C03629=1083.943,283.313,-84.249,175.955,24.447,154.018
C03630=1083.938,283.065,-84.220,175.952,24.443,154.018
C03631=1083.932,282.817,-84.190,175.949,24.440,154.017
C03632=1083.926,282.569,-84.160,175.947,24.436,154.017
C03633=1083.920,282.321,-84.131,175.944,24.433,154.016
C03634=1083.915,282.073,-84.101,175.941,24.429,154.016
C03635=1083.910,281.824,-84.072,175.938,24.426,154.015
C03636=1083.903,281.576,-84.043,175.936,24.423,154.015
C03637=1083.898,281.328,-84.013,175.933,24.419,154.015
C03638=1083.892,281.079,-83.984,175.930,24.415,154.014
C03639=1083.886,280.831,-83.954,175.927,24.412,154.014
C03640=1083.881,280.584,-83.925,175.925,24.409,154.013
C03641=1083.875,280.335,-83.896,175.922,24.405,154.013
C03642=1083.870,280.087,-83.867,175.919,24.402,154.013
C03643=1083.863,279.839,-83.837,175.916,24.398,154.012
C03644=1083.858,279.590,-83.808,175.913,24.395,154.012
C03645=1083.852,279.342,-83.778,175.910,24.391,154.011
C03646=1083.846,279.094,-83.749,175.907,24.388,154.011
C03647=1083.841,278.846,-83.720,175.904,24.384,154.011
C03648=1083.835,278.598,-83.691,175.902,24.381,154.010
C03649=1083.829,278.350,-83.661,175.899,24.378,154.010
C03650=1083.823,278.101,-83.632,175.896,24.374,154.009
C03651=1083.818,277.853,-83.603,175.893,24.370,154.009
C03652=1083.812,277.606,-83.574,175.891,24.367,154.009
C03653=1083.807,277.356,-83.545,175.888,24.364,154.008
C03654=1083.800,277.108,-83.516,175.885,24.360,154.008
C03655=1083.791,276.725,-83.471,175.881,24.355,154.007
C03656=1083.783,276.341,-83.426,175.877,24.350,154.007
C03657=1083.773,275.957,-83.380,175.872,24.345,154.006
C03658=1083.765,275.574,-83.336,175.868,24.339,154.005
C03659=1083.760,275.325,-83.307,175.865,24.336,154.005
C03660=1083.753,275.077,-83.278,175.863,24.333,154.005
C03661=1083.748,274.829,-83.249,175.860,24.329,154.004
C03662=1083.743,274.581,-83.221,175.857,24.325,154.004
C03663=1083.736,274.333,-83.192,175.854,24.322,154.003
C03664=1083.731,274.084,-83.162,175.852,24.319,154.003
C03665=1083.726,273.836,-83.134,175.849,24.315,154.003
C03666=1083.719,273.588,-83.105,175.846,24.312,154.002
C03667=1083.714,273.339,-83.075,175.843,24.309,154.002
C03668=1083.708,273.091,-83.047,175.840,24.305,154.001
C03669=1083.702,272.843,-83.018,175.837,24.302,154.001
C03670=1083.697,272.594,-82.989,175.835,24.299,154.001
C03671=1083.691,272.346,-82.960,175.832,24.295,154.000
C03672=1083.685,272.099,-82.932,175.829,24.291,154.000
C03673=1083.679,271.850,-82.903,175.826,24.288,153.999
C03674=1083.674,271.601,-82.874,175.824,24.285,153.999
C03675=1083.668,271.353,-82.846,175.821,24.282,153.999
C03676=1083.662,271.105,-82.817,175.818,24.278,153.998
C03677=1083.656,270.857,-82.788,175.816,24.275,153.998
C03678=1083.651,270.609,-82.760,175.813,24.271,153.998
C03679=1083.645,270.360,-82.731,175.810,24.268,153.997
C03680=1083.639,270.111,-82.702,175.808,24.265,153.997
C03681=1083.634,269.864,-82.674,175.804,24.262,153.996
C03682=1083.628,269.615,-82.645,175.801,24.258,153.996
C03683=1083.621,269.367,-82.616,175.799,24.255,153.996
C03684=1083.617,269.119,-82.588,175.796,24.251,153.995
C03685=1083.611,268.870,-82.560,175.793,24.248,153.995
C03686=1083.605,268.622,-82.531,175.791,24.245,153.995
C03687=1083.599,268.374,-82.503,175.788,24.241,153.994
C03688=1083.593,268.125,-82.474,175.785,24.238,153.994
C03689=1083.588,267.878,-82.446,175.782,24.234,153.993
C03690=1083.582,267.629,-82.417,175.780,24.231,153.993
C03691=1083.576,267.381,-82.389,175.777,24.228,153.993
C03692=1083.570,267.132,-82.361,175.774,24.224,153.992
C03693=1083.564,266.884,-82.332,175.772,24.221,153.992
C03694=1083.559,266.636,-82.304,175.769,24.218,153.991
C03695=1083.553,266.387,-82.276,175.766,24.215,153.991
C03696=1083.548,266.139,-82.248,175.763,24.211,153.991
C03697=1083.542,265.891,-82.218,175.760,24.208,153.990
C03698=1083.537,265.642,-82.190,175.758,24.205,153.990
C03699=1083.531,265.394,-82.162,175.755,24.201,153.990
C03700=1083.525,265.146,-82.134,175.752,24.198,153.989
C03701=1083.520,264.897,-82.105,175.750,24.195,153.989
C03702=1083.514,264.649,-82.077,175.747,24.191,153.988
C03703=1083.508,264.400,-82.049,175.744,24.188,153.988
C03704=1083.503,264.153,-82.020,175.742,24.184,153.988
C03705=1083.497,263.904,-81.992,175.739,24.181,153.987
C03706=1083.490,263.656,-81.964,175.736,24.178,153.987
C03707=1083.482,263.274,-81.921,175.732,24.173,153.987
C03708=1083.473,262.894,-81.878,175.728,24.168,153.986
C03709=1083.464,262.513,-81.836,175.724,24.164,153.985
C03710=1083.455,262.133,-81.793,175.719,24.158,153.985
C03711=1083.449,261.884,-81.764,175.716,24.155,153.984
C03712=1083.444,261.636,-81.736,175.714,24.152,153.984
C03713=1083.437,261.387,-81.709,175.711,24.148,153.984
C03714=1083.431,261.139,-81.681,175.709,24.146,153.983
C03715=1083.426,260.890,-81.652,175.706,24.142,153.983
C03716=1083.419,260.643,-81.625,175.703,24.138,153.983
C03717=1083.414,260.393,-81.597,175.701,24.136,153.982
C03718=1083.408,260.145,-81.570,175.698,24.132,153.982
C03719=1083.403,259.897,-81.541,175.695,24.129,153.982
C03720=1083.396,259.649,-81.514,175.692,24.126,153.981
C03721=1083.391,259.400,-81.486,175.689,24.122,153.981
C03722=1083.385,259.152,-81.458,175.687,24.120,153.981
C03723=1083.379,258.903,-81.431,175.684,24.116,153.980
C03724=1083.373,258.655,-81.403,175.681,24.112,153.980
C03725=1083.368,258.407,-81.375,175.679,24.110,153.980
C03726=1083.362,258.158,-81.346,175.676,24.106,153.979
C03727=1083.356,257.910,-81.319,175.674,24.103,153.979
C03728=1083.350,257.661,-81.291,175.671,24.100,153.978
C03729=1083.345,257.413,-81.263,175.668,24.096,153.978
C03730=1083.339,257.165,-81.236,175.666,24.093,153.978
C03731=1083.333,256.916,-81.208,175.663,24.090,153.977
C03732=1083.328,256.668,-81.180,175.660,24.087,153.977
C03733=1083.321,256.419,-81.153,175.657,24.083,153.977
C03734=1083.316,256.171,-81.125,175.654,24.080,153.976
C03735=1083.310,255.923,-81.098,175.652,24.077,153.976
C03736=1083.304,255.674,-81.070,175.649,24.074,153.976
C03737=1083.299,255.426,-81.043,175.647,24.071,153.975
C03738=1083.293,255.178,-81.015,175.644,24.067,153.975
C03739=1083.288,254.928,-80.988,175.641,24.064,153.975
C03740=1083.282,254.680,-80.960,175.639,24.061,153.974
C03741=1083.276,254.433,-80.932,175.636,24.057,153.974
C03742=1083.270,254.183,-80.905,175.634,24.055,153.973
C03743=1083.264,253.936,-80.877,175.631,24.051,153.973
C03744=1083.259,253.687,-80.850,175.628,24.048,153.973
C03745=1083.253,253.438,-80.822,175.625,24.045,153.972
C03746=1083.248,253.190,-80.795,175.622,24.041,153.972
C03747=1083.242,252.942,-80.767,175.620,24.038,153.972
C03748=1083.237,252.693,-80.740,175.617,24.035,153.971
C03749=1083.231,252.445,-80.712,175.615,24.032,153.971
C03750=1083.226,252.196,-80.685,175.612,24.028,153.971
C03751=1083.220,251.948,-80.658,175.610,24.025,153.970
C03752=1083.214,251.699,-80.630,175.607,24.022,153.970
C03753=1083.208,251.450,-80.603,175.604,24.018,153.969
C03754=1083.203,251.202,-80.575,175.602,24.015,153.969
C03755=1083.197,250.954,-80.549,175.599,24.012,153.969
C03756=1083.192,250.705,-80.521,175.597,24.009,153.968
C03757=1083.186,250.458,-80.494,175.594,24.005,153.968
C03758=1083.180,250.208,-80.466,175.591,24.002,153.968
C03759=1083.172,249.825,-80.424,175.587,23.997,153.967
C03760=1083.163,249.441,-80.383,175.583,23.992,153.966
C03761=1083.155,249.058,-80.341,175.579,23.987,153.966
C03762=1083.146,248.674,-80.299,175.575,23.982,153.965
C03763=1083.140,248.426,-80.272,175.572,23.978,153.965
C03764=1083.135,248.177,-80.245,175.570,23.975,153.965
C03765=1083.129,247.929,-80.217,175.567,23.972,153.964
C03766=1083.123,247.680,-80.190,175.565,23.969,153.964
C03767=1083.118,247.432,-80.163,175.562,23.965,153.964
C03768=1083.113,247.183,-80.136,175.560,23.963,153.963
C03769=1083.107,246.935,-80.109,175.557,23.959,153.963
C03770=1083.101,246.686,-80.082,175.555,23.956,153.962
C03771=1083.096,246.438,-80.054,175.551,23.953,153.962
C03772=1083.089,246.189,-80.027,175.549,23.949,153.962
C03773=1083.084,245.941,-80.001,175.546,23.946,153.961
C03774=1083.079,245.692,-79.974,175.543,23.943,153.961
C03775=1083.073,245.444,-79.947,175.541,23.939,153.961
C03776=1083.067,245.195,-79.920,175.538,23.936,153.960
C03777=1083.062,244.947,-79.893,175.536,23.933,153.960
C03778=1083.056,244.698,-79.866,175.533,23.930,153.960
C03779=1083.050,244.450,-79.840,175.531,23.927,153.959
C03780=1083.045,244.202,-79.813,175.528,23.923,153.959
C03781=1083.039,243.952,-79.785,175.526,23.921,153.959
C03782=1083.033,243.704,-79.759,175.523,23.917,153.958
C03783=1083.028,243.455,-79.732,175.521,23.914,153.958
C03784=1083.022,243.207,-79.706,175.517,23.911,153.958
C03785=1083.017,242.958,-79.678,175.515,23.907,153.957
C03786=1083.011,242.710,-79.652,175.512,23.904,153.957
C03787=1083.005,242.462,-79.625,175.510,23.901,153.956
C03788=1082.999,242.213,-79.598,175.507,23.897,153.956
C03789=1082.994,241.965,-79.572,175.505,23.895,153.956
C03790=1082.988,241.716,-79.546,175.502,23.891,153.955
C03791=1082.982,241.468,-79.519,175.500,23.888,153.955
C03792=1082.976,241.219,-79.492,175.497,23.885,153.955
C03793=1082.970,240.970,-79.465,175.495,23.882,153.954
C03794=1082.964,240.722,-79.439,175.492,23.878,153.954
C03795=1082.959,240.473,-79.412,175.489,23.876,153.954
C03796=1082.954,240.224,-79.386,175.486,23.872,153.953
C03797=1082.948,239.976,-79.359,175.484,23.869,153.953
C03798=1082.942,239.728,-79.332,175.481,23.866,153.953
C03799=1082.937,239.479,-79.306,175.479,23.863,153.952
C03800=1082.931,239.230,-79.280,175.476,23.859,153.952
C03801=1082.925,238.982,-79.253,175.474,23.857,153.952
C03802=1082.920,238.733,-79.226,175.471,23.853,153.951
C03803=1082.914,238.485,-79.200,175.469,23.850,153.951
C03804=1082.908,238.236,-79.174,175.467,23.847,153.951
C03805=1082.903,237.988,-79.147,175.464,23.844,153.950
C03806=1082.897,237.739,-79.121,175.461,23.841,153.950
C03807=1082.891,237.490,-79.095,175.459,23.837,153.950
C03808=1082.886,237.242,-79.068,175.456,23.835,153.949
C03809=1082.880,236.993,-79.042,175.453,23.831,153.949
C03810=1082.874,236.745,-79.015,175.451,23.828,153.949
C03811=1082.866,236.354,-78.975,175.447,23.823,153.948
C03812=1082.856,235.964,-78.933,175.443,23.818,153.947
C03813=1082.847,235.574,-78.892,175.439,23.813,153.947
C03814=1082.839,235.183,-78.851,175.435,23.808,153.946
C03815=1082.832,234.935,-78.825,175.433,23.805,153.946
C03816=1082.827,234.686,-78.799,175.430,23.801,153.946
C03817=1082.821,234.438,-78.772,175.428,23.799,153.945
C03818=1082.816,234.189,-78.746,175.425,23.795,153.945
C03819=1082.810,233.940,-78.719,175.423,23.792,153.945
C03820=1082.805,233.692,-78.693,175.419,23.789,153.944
C03821=1082.799,233.443,-78.667,175.417,23.786,153.944
C03822=1082.794,233.195,-78.641,175.414,23.782,153.944
C03823=1082.788,232.946,-78.616,175.412,23.779,153.943
C03824=1082.782,232.698,-78.589,175.410,23.776,153.943
C03825=1082.776,232.449,-78.563,175.407,23.773,153.943
C03826=1082.771,232.201,-78.537,175.405,23.770,153.942
C03827=1082.765,231.952,-78.511,175.402,23.766,153.942
C03828=1082.759,231.703,-78.485,175.400,23.764,153.942
C03829=1082.753,231.454,-78.459,175.397,23.760,153.941
C03830=1082.748,231.206,-78.433,175.395,23.757,153.941
C03831=1082.743,230.957,-78.407,175.392,23.754,153.941
C03832=1082.737,230.708,-78.381,175.390,23.751,153.940
C03833=1082.731,230.460,-78.355,175.387,23.748,153.940
C03834=1082.725,230.211,-78.329,175.384,23.744,153.940
C03835=1082.720,229.962,-78.303,175.382,23.741,153.939
C03836=1082.714,229.715,-78.278,175.379,23.738,153.939
C03837=1082.709,229.466,-78.252,175.377,23.735,153.939
C03838=1082.703,229.217,-78.226,175.375,23.732,153.938
C03839=1082.697,228.968,-78.200,175.372,23.729,153.938
C03840=1082.691,228.719,-78.175,175.370,23.726,153.937
C03841=1082.685,228.471,-78.148,175.367,23.722,153.937
C03842=1082.679,228.222,-78.123,175.365,23.719,153.937
C03843=1082.675,227.974,-78.097,175.362,23.716,153.937
C03844=1082.668,227.725,-78.072,175.359,23.713,153.936
C03845=1082.663,227.476,-78.046,175.357,23.710,153.936
C03846=1082.657,227.228,-78.020,175.354,23.707,153.936
C03847=1082.651,226.979,-77.994,175.352,23.704,153.935
C03848=1082.646,226.731,-77.969,175.350,23.701,153.935
C03849=1082.640,226.482,-77.943,175.347,23.697,153.935
C03850=1082.634,226.233,-77.917,175.345,23.694,153.934
C03851=1082.628,225.985,-77.892,175.342,23.691,153.934
C03852=1082.623,225.736,-77.866,175.340,23.688,153.933
C03853=1082.617,225.488,-77.841,175.338,23.685,153.933
C03854=1082.612,225.239,-77.815,175.335,23.681,153.933
C03855=1082.605,224.990,-77.789,175.332,23.679,153.932
C03856=1082.601,224.742,-77.764,175.329,23.675,153.932
C03857=1082.594,224.493,-77.738,175.327,23.672,153.932
C03858=1082.589,224.244,-77.713,175.325,23.669,153.931
C03859=1082.583,223.996,-77.688,175.322,23.666,153.931
C03860=1082.578,223.747,-77.662,175.320,23.663,153.931
C03861=1082.572,223.499,-77.636,175.318,23.660,153.930
C03862=1082.566,223.249,-77.611,175.315,23.656,153.930
C03863=1082.557,222.851,-77.570,175.311,23.651,153.929
C03864=1082.549,222.452,-77.529,175.307,23.646,153.929
C03865=1082.540,222.053,-77.489,175.303,23.641,153.928
C03866=1082.530,221.654,-77.448,175.300,23.636,153.928
C03867=1082.525,221.406,-77.423,175.297,23.633,153.928
C03868=1082.519,221.157,-77.397,175.294,23.630,153.927
C03869=1082.513,220.907,-77.372,175.292,23.627,153.927
C03870=1082.508,220.660,-77.347,175.289,23.624,153.927
C03871=1082.501,220.411,-77.322,175.287,23.621,153.926
C03872=1082.496,220.162,-77.296,175.284,23.618,153.926
C03873=1082.491,219.913,-77.272,175.282,23.614,153.926
C03874=1082.484,219.665,-77.246,175.280,23.612,153.925
C03875=1082.479,219.416,-77.221,175.277,23.608,153.925
C03876=1082.473,219.168,-77.196,175.275,23.605,153.925
C03877=1082.468,218.918,-77.171,175.273,23.602,153.924
C03878=1082.461,218.670,-77.146,175.270,23.599,153.924
C03879=1082.456,218.421,-77.120,175.268,23.596,153.924
C03880=1082.451,218.172,-77.095,175.265,23.593,153.923
C03881=1082.445,217.924,-77.070,175.263,23.589,153.923
C03882=1082.439,217.676,-77.045,175.260,23.586,153.923
C03883=1082.434,217.426,-77.020,175.258,23.583,153.922
C03884=1082.428,217.178,-76.995,175.255,23.580,153.922
C03885=1082.422,216.929,-76.970,175.253,23.577,153.921
C03886=1082.416,216.681,-76.945,175.251,23.574,153.921
C03887=1082.411,216.432,-76.919,175.248,23.570,153.921
C03888=1082.406,216.183,-76.895,175.246,23.568,153.921
C03889=1082.399,215.934,-76.870,175.244,23.564,153.920
C03890=1082.394,215.685,-76.845,175.241,23.561,153.920
C03891=1082.388,215.437,-76.820,175.239,23.558,153.919
C03892=1082.383,215.188,-76.795,175.236,23.555,153.919
C03893=1082.377,214.940,-76.770,175.234,23.552,153.919
C03894=1082.371,214.690,-76.745,175.231,23.549,153.919
C03895=1082.366,214.442,-76.720,175.229,23.546,153.918
C03896=1082.360,214.193,-76.696,175.226,23.542,153.918
C03897=1082.355,213.945,-76.670,175.224,23.539,153.917
C03898=1082.349,213.696,-76.646,175.222,23.536,153.917
C03899=1082.343,213.448,-76.621,175.219,23.533,153.917
C03900=1082.338,213.198,-76.596,175.217,23.530,153.916
C03901=1082.332,212.950,-76.572,175.215,23.527,153.916
C03902=1082.326,212.701,-76.546,175.212,23.523,153.916
C03903=1082.321,212.452,-76.522,175.210,23.520,153.915
C03904=1082.315,212.204,-76.497,175.208,23.517,153.915
C03905=1082.309,211.955,-76.473,175.205,23.514,153.915
C03906=1082.303,211.706,-76.448,175.203,23.511,153.914
C03907=1082.298,211.458,-76.423,175.200,23.508,153.914
C03908=1082.293,211.208,-76.398,175.198,23.505,153.914
C03909=1082.287,210.960,-76.373,175.195,23.502,153.913
C03910=1082.282,210.711,-76.349,175.193,23.498,153.913
C03911=1082.276,210.462,-76.324,175.191,23.496,153.913
C03912=1082.270,210.214,-76.300,175.188,23.492,153.912
C03913=1082.264,209.965,-76.276,175.186,23.489,153.912
C03914=1082.258,209.717,-76.251,175.184,23.486,153.912
C03915=1082.250,209.321,-76.212,175.180,23.481,153.911
C03916=1082.241,208.926,-76.173,175.176,23.476,153.911
C03917=1082.232,208.532,-76.134,175.172,23.471,153.910
C03918=1082.222,208.137,-76.095,175.169,23.466,153.910
C03919=1082.199,207.105,-75.995,175.076,23.417,153.912
C03920=1082.193,206.857,-75.972,175.073,23.415,153.912
C03921=1082.188,206.608,-75.947,175.071,23.413,153.912
C03922=1082.182,206.358,-75.923,175.068,23.411,153.911
C03923=1082.176,206.110,-75.900,175.065,23.408,153.911
C03924=1082.171,205.861,-75.875,175.063,23.406,153.911
C03925=1082.166,205.612,-75.852,175.060,23.404,153.911
C03926=1082.160,205.364,-75.828,175.058,23.402,153.911
C03927=1082.155,205.115,-75.804,175.056,23.399,153.911
C03928=1082.149,204.866,-75.779,175.053,23.397,153.911
C03929=1082.143,204.617,-75.756,175.051,23.395,153.911
C03930=1082.138,204.369,-75.732,175.048,23.393,153.910
C03931=1082.132,204.120,-75.708,175.046,23.391,153.910
C03932=1082.127,203.871,-75.685,175.044,23.389,153.910
C03933=1082.121,203.623,-75.661,175.040,23.386,153.910
C03934=1082.116,203.373,-75.637,175.038,23.384,153.910
C03935=1082.110,203.124,-75.613,175.036,23.382,153.910
C03936=1082.104,202.876,-75.589,175.033,23.380,153.910
C03937=1082.099,202.627,-75.566,175.031,23.378,153.910
C03938=1082.093,202.378,-75.542,175.028,23.375,153.910
C03939=1082.088,202.129,-75.519,175.026,23.373,153.909
C03940=1082.082,201.880,-75.494,175.024,23.371,153.909
C03941=1082.076,201.631,-75.471,175.021,23.369,153.909
C03942=1082.070,201.383,-75.447,175.019,23.367,153.909
C03943=1082.065,201.134,-75.424,175.016,23.365,153.909
C03944=1082.059,200.885,-75.400,175.014,23.363,153.909
C03945=1082.054,200.636,-75.377,175.012,23.361,153.909
C03946=1082.048,200.388,-75.353,175.009,23.358,153.909
C03947=1082.042,200.138,-75.330,175.006,23.356,153.909
C03948=1082.036,199.890,-75.306,175.003,23.354,153.909
C03949=1082.031,199.641,-75.283,175.001,23.352,153.908
C03950=1082.025,199.393,-75.259,174.999,23.350,153.908
C03951=1082.020,199.143,-75.235,174.996,23.348,153.908
C03952=1082.014,198.894,-75.212,174.994,23.346,153.908
C03953=1082.008,198.646,-75.189,174.992,23.343,153.908
C03954=1082.003,198.397,-75.165,174.989,23.342,153.908
C03955=1081.996,198.148,-75.141,174.987,23.339,153.908
C03956=1081.990,197.899,-75.118,174.984,23.337,153.908
C03957=1081.985,197.650,-75.095,174.982,23.335,153.908
C03958=1081.979,197.402,-75.071,174.979,23.333,153.907
C03959=1081.974,197.153,-75.048,174.977,23.331,153.907
C03960=1081.969,196.904,-75.025,174.975,23.329,153.907
C03961=1081.963,196.655,-75.001,174.972,23.327,153.907
C03962=1081.957,196.406,-74.978,174.970,23.325,153.907
C03963=1081.952,196.157,-74.954,174.967,23.322,153.907
C03964=1081.946,195.909,-74.931,174.965,23.320,153.907
C03965=1081.940,195.660,-74.908,174.963,23.319,153.907
C03966=1081.935,195.411,-74.884,174.960,23.316,153.907
C03967=1081.929,195.162,-74.861,174.958,23.314,153.906
C03968=1081.923,194.914,-74.838,174.956,23.312,153.906
C03969=1081.918,194.665,-74.815,174.953,23.310,153.906
C03970=1081.913,194.415,-74.791,174.951,23.308,153.906
C03971=1081.907,194.167,-74.768,174.948,23.306,153.906
C03972=1081.901,193.918,-74.745,174.946,23.303,153.906
C03973=1081.896,193.669,-74.721,174.944,23.301,153.906
C03974=1081.890,193.420,-74.698,174.941,23.299,153.906
C03975=1081.884,193.171,-74.675,174.939,23.297,153.906
C03976=1081.879,192.922,-74.652,174.936,23.295,153.905
C03977=1081.874,192.673,-74.629,174.934,23.293,153.905
C03978=1081.868,192.424,-74.606,174.932,23.291,153.905
C03979=1081.862,192.175,-74.583,174.929,23.289,153.905
C03980=1081.856,191.897,-74.556,174.926,23.286,153.905
C03981=1081.850,191.617,-74.531,174.924,23.284,153.905
C03982=1081.843,191.338,-74.505,174.921,23.281,153.905
C03983=1081.837,191.058,-74.479,174.918,23.279,153.905
C03984=1081.832,190.810,-74.456,174.916,23.277,153.904
C03985=1081.827,190.560,-74.433,174.913,23.274,153.904
C03986=1081.821,190.312,-74.409,174.911,23.272,153.904
C03987=1081.815,190.064,-74.386,174.909,23.270,153.904
C03988=1081.810,189.815,-74.363,174.906,23.268,153.904
C03989=1081.804,189.566,-74.340,174.905,23.266,153.904
C03990=1081.799,189.317,-74.317,174.902,23.264,153.904
C03991=1081.794,189.067,-74.295,174.900,23.262,153.903
C03992=1081.788,188.818,-74.272,174.898,23.259,153.903
C03993=1081.782,188.570,-74.249,174.895,23.257,153.903
C03994=1081.776,188.321,-74.226,174.893,23.255,153.903
C03995=1081.771,188.072,-74.203,174.890,23.253,153.903
C03996=1081.766,187.823,-74.180,174.888,23.251,153.903
C03997=1081.761,187.574,-74.157,174.886,23.249,153.903
C03998=1081.755,187.325,-74.134,174.883,23.246,153.903
C03999=1081.749,187.077,-74.111,174.881,23.244,153.902
C04000=1081.744,186.828,-74.088,174.879,23.242,153.902
C04001=1081.738,186.579,-74.065,174.876,23.240,153.902
C04002=1081.733,186.330,-74.042,174.874,23.238,153.902
C04003=1081.728,186.081,-74.020,174.871,23.236,153.902
C04004=1081.722,185.832,-73.997,174.869,23.233,153.902
C04005=1081.717,185.584,-73.974,174.867,23.231,153.902
C04006=1081.711,185.335,-73.951,174.864,23.229,153.902
C04007=1081.705,185.086,-73.928,174.862,23.227,153.901
C04008=1081.700,184.836,-73.906,174.860,23.224,153.901
C04009=1081.694,184.587,-73.883,174.858,23.223,153.901
C04010=1081.689,184.339,-73.860,174.856,23.221,153.901
C04011=1081.683,184.090,-73.837,174.853,23.219,153.901
C04012=1081.677,183.840,-73.815,174.851,23.217,153.901
C04013=1081.672,183.592,-73.793,174.849,23.215,153.901
C04014=1081.666,183.343,-73.770,174.846,23.212,153.901
C04015=1081.660,183.094,-73.747,174.844,23.211,153.901
C04016=1081.654,182.845,-73.725,174.841,23.208,153.901
C04017=1081.648,182.596,-73.702,174.839,23.206,153.900
C04018=1081.642,182.347,-73.679,174.836,23.204,153.900
C04019=1081.637,182.098,-73.657,174.834,23.202,153.900
C04020=1081.631,181.850,-73.635,174.832,23.200,153.900
C04021=1081.625,181.601,-73.612,174.830,23.199,153.900
C04022=1081.620,181.352,-73.590,174.828,23.196,153.900
C04023=1081.614,181.103,-73.567,174.825,23.194,153.900
C04024=1081.608,180.854,-73.545,174.823,23.192,153.900
C04025=1081.602,180.605,-73.522,174.821,23.190,153.900
C04026=1081.597,180.356,-73.500,174.818,23.188,153.899
C04027=1081.591,180.107,-73.478,174.816,23.186,153.899
C04028=1081.585,179.858,-73.455,174.813,23.184,153.899
C04029=1081.580,179.609,-73.432,174.811,23.182,153.899
C04030=1081.574,179.360,-73.410,174.809,23.179,153.899
C04031=1081.568,179.112,-73.388,174.807,23.178,153.899
C04032=1081.563,178.863,-73.366,174.805,23.176,153.899
C04033=1081.557,178.614,-73.343,174.802,23.173,153.899
C04034=1081.551,178.364,-73.321,174.800,23.171,153.899
C04035=1081.546,178.116,-73.299,174.798,23.169,153.899
C04036=1081.540,177.867,-73.277,174.795,23.167,153.898
C04037=1081.534,177.618,-73.254,174.793,23.165,153.898
C04038=1081.529,177.369,-73.232,174.791,23.163,153.898
C04039=1081.523,177.120,-73.209,174.789,23.161,153.898
C04040=1081.517,176.871,-73.188,174.787,23.159,153.898
C04041=1081.512,176.622,-73.165,174.784,23.157,153.898
C04042=1081.506,176.373,-73.143,174.782,23.155,153.898
C04043=1081.501,176.124,-73.121,174.779,23.153,153.898
C04044=1081.494,175.845,-73.096,174.777,23.151,153.897
C04045=1081.488,175.565,-73.071,174.775,23.148,153.897
C04046=1081.482,175.285,-73.046,174.771,23.146,153.897
C04047=1081.475,175.006,-73.021,174.769,23.143,153.897
C04048=1081.470,174.757,-72.999,174.767,23.141,153.897
C04049=1081.464,174.508,-72.977,174.764,23.139,153.897
C04050=1081.458,174.259,-72.954,174.763,23.137,153.897
C04051=1081.453,174.010,-72.932,174.761,23.135,153.896
C04052=1081.447,173.761,-72.911,174.758,23.133,153.896
C04053=1081.442,173.512,-72.888,174.756,23.131,153.896
C04054=1081.436,173.263,-72.866,174.753,23.128,153.896
C04055=1081.431,173.014,-72.844,174.751,23.126,153.896
C04056=1081.425,172.765,-72.822,174.750,23.124,153.896
C04057=1081.419,172.517,-72.800,174.747,23.122,153.896
C04058=1081.414,172.267,-72.778,174.745,23.120,153.896
C04059=1081.408,172.018,-72.756,174.743,23.118,153.896
C04060=1081.403,171.770,-72.734,174.740,23.116,153.895
C04061=1081.397,171.520,-72.712,174.738,23.114,153.895
C04062=1081.391,171.271,-72.690,174.736,23.112,153.895
C04063=1081.386,171.022,-72.668,174.734,23.109,153.895
C04064=1081.380,170.774,-72.646,174.732,23.108,153.895
C04065=1081.375,170.525,-72.624,174.729,23.105,153.895
C04066=1081.369,170.276,-72.602,174.727,23.103,153.895
C04067=1081.364,170.027,-72.580,174.725,23.101,153.895
C04068=1081.359,169.777,-72.558,174.723,23.099,153.894
C04069=1081.352,169.528,-72.536,174.721,23.097,153.894
C04070=1081.348,169.279,-72.515,174.718,23.094,153.894
C04071=1081.341,169.031,-72.492,174.716,23.092,153.894
C04072=1081.336,168.782,-72.470,174.714,23.090,153.894
C04073=1081.330,168.533,-72.449,174.712,23.089,153.894
C04074=1081.325,168.284,-72.427,174.710,23.086,153.894
C04075=1081.319,168.035,-72.405,174.707,23.084,153.893
C04076=1081.314,167.786,-72.383,174.705,23.082,153.893
C04077=1081.308,167.537,-72.362,174.703,23.080,153.893
C04078=1081.303,167.288,-72.340,174.700,23.077,153.893
C04079=1081.297,167.039,-72.318,174.699,23.075,153.893
C04080=1081.292,166.790,-72.296,174.697,23.073,153.893
C04081=1081.287,166.540,-72.274,174.694,23.071,153.893
C04082=1081.281,166.292,-72.253,174.692,23.069,153.892
C04083=1081.276,166.042,-72.231,174.690,23.066,153.892
C04084=1081.270,165.794,-72.209,174.688,23.065,153.892
C04085=1081.265,165.544,-72.187,174.686,23.062,153.892
C04086=1081.259,165.296,-72.166,174.684,23.060,153.892
C04087=1081.253,165.047,-72.144,174.681,23.058,153.892
C04088=1081.248,164.798,-72.122,174.680,23.056,153.892
C04089=1081.243,164.549,-72.101,174.677,23.054,153.891
C04090=1081.237,164.300,-72.079,174.675,23.052,153.891
C04091=1081.232,164.051,-72.058,174.673,23.050,153.891
C04092=1081.226,163.802,-72.035,174.670,23.047,153.891
C04093=1081.221,163.553,-72.014,174.669,23.045,153.891
C04094=1081.215,163.304,-71.992,174.666,23.043,153.891
C04095=1081.210,163.055,-71.971,174.664,23.041,153.891
C04096=1081.205,162.806,-71.950,174.662,23.039,153.890
C04097=1081.199,162.557,-71.928,174.660,23.037,153.890
C04098=1081.194,162.308,-71.906,174.658,23.035,153.890
C04099=1081.188,162.059,-71.884,174.656,23.032,153.890
C04100=1081.183,161.810,-71.863,174.653,23.030,153.890
C04101=1081.178,161.561,-71.841,174.651,23.028,153.890
C04102=1081.172,161.311,-71.820,174.650,23.026,153.890
C04103=1081.166,161.063,-71.799,174.647,23.024,153.889
C04104=1081.161,160.813,-71.777,174.645,23.021,153.889
C04105=1081.155,160.565,-71.756,174.643,23.019,153.889
C04106=1081.149,160.316,-71.734,174.641,23.017,153.889
C04107=1081.144,160.067,-71.713,174.639,23.015,153.889
C04108=1081.137,159.787,-71.689,174.637,23.013,153.889
C04109=1081.131,159.507,-71.665,174.634,23.010,153.889
C04110=1081.125,159.227,-71.641,174.632,23.008,153.888
C04111=1081.119,158.947,-71.617,174.630,23.006,153.888
C04112=1081.113,158.698,-71.596,174.627,23.004,153.888
C04113=1081.107,158.449,-71.575,174.625,23.001,153.888
C04114=1081.101,158.200,-71.554,174.623,22.999,153.888
C04115=1081.096,157.951,-71.532,174.621,22.997,153.888
C04116=1081.091,157.702,-71.511,174.619,22.995,153.888
C04117=1081.085,157.452,-71.489,174.616,22.993,153.887
C04118=1081.079,157.204,-71.468,174.614,22.990,153.887
C04119=1081.074,156.954,-71.447,174.612,22.989,153.887
C04120=1081.068,156.706,-71.426,174.610,22.987,153.887
C04121=1081.063,156.457,-71.405,174.608,22.984,153.887
C04122=1081.057,156.207,-71.384,174.605,22.982,153.887
C04123=1081.051,155.959,-71.363,174.604,22.980,153.887
C04124=1081.047,155.709,-71.341,174.602,22.978,153.886
C04125=1081.040,155.460,-71.320,174.599,22.976,153.886
C04126=1081.035,155.212,-71.298,174.598,22.974,153.886
C04127=1081.030,154.963,-71.278,174.596,22.972,153.886
C04128=1081.023,154.713,-71.256,174.593,22.969,153.886
C04129=1081.018,154.464,-71.236,174.591,22.967,153.886
C04130=1081.012,154.215,-71.214,174.590,22.965,153.886
C04131=1081.007,153.966,-71.194,174.587,22.963,153.885
C04132=1081.001,153.717,-71.172,174.585,22.961,153.885
C04133=1080.995,153.468,-71.151,174.583,22.959,153.885
C04134=1080.990,153.219,-71.130,174.581,22.957,153.885
C04135=1080.985,152.970,-71.110,174.579,22.955,153.885
C04136=1080.978,152.721,-71.088,174.576,22.953,153.885
C04137=1080.973,152.472,-71.067,174.575,22.951,153.885
C04138=1080.968,152.223,-71.046,174.573,22.948,153.885
C04139=1080.962,151.974,-71.026,174.570,22.946,153.884
C04140=1080.956,151.724,-71.005,174.569,22.944,153.884
C04141=1080.950,151.476,-70.984,174.566,22.942,153.884
C04142=1080.945,151.227,-70.963,174.564,22.940,153.884
C04143=1080.939,150.978,-70.942,174.562,22.937,153.884
C04144=1080.933,150.728,-70.921,174.560,22.936,153.884
C04145=1080.928,150.479,-70.901,174.558,22.933,153.883
C04146=1080.923,150.231,-70.879,174.556,22.931,153.883
C04147=1080.917,149.981,-70.858,174.554,22.929,153.883
C04148=1080.912,149.732,-70.838,174.552,22.927,153.883
C04149=1080.906,149.483,-70.817,174.550,22.925,153.883
C04150=1080.900,149.234,-70.796,174.548,22.923,153.883
C04151=1080.895,148.984,-70.775,174.546,22.920,153.883
C04152=1080.889,148.736,-70.754,174.544,22.918,153.882
C04153=1080.883,148.487,-70.734,174.542,22.916,153.882
C04154=1080.877,148.237,-70.713,174.540,22.914,153.882
C04155=1080.872,147.989,-70.692,174.537,22.912,153.882
C04156=1080.867,147.740,-70.671,174.536,22.910,153.882
C04157=1080.861,147.491,-70.651,174.534,22.908,153.882
C04158=1080.855,147.241,-70.630,174.531,22.905,153.882
C04159=1080.849,146.993,-70.609,174.530,22.903,153.881
C04160=1080.844,146.743,-70.588,174.528,22.901,153.881
C04161=1080.839,146.494,-70.568,174.525,22.899,153.881
C04162=1080.832,146.245,-70.548,174.524,22.897,153.881
C04163=1080.827,145.996,-70.526,174.521,22.895,153.881
C04164=1080.821,145.747,-70.506,174.519,22.893,153.881
C04165=1080.816,145.498,-70.485,174.518,22.891,153.881
C04166=1080.809,145.249,-70.465,174.515,22.889,153.880
C04167=1080.804,144.999,-70.444,174.513,22.887,153.880
C04168=1080.799,144.750,-70.424,174.512,22.885,153.880
C04169=1080.793,144.502,-70.403,174.509,22.882,153.880
C04170=1080.787,144.253,-70.383,174.507,22.880,153.880
C04171=1080.782,144.003,-70.362,174.505,22.878,153.880
C04172=1080.775,143.723,-70.340,174.503,22.875,153.879
C04173=1080.769,143.443,-70.316,174.501,22.873,153.879
C04174=1080.763,143.164,-70.293,174.499,22.871,153.879
C04175=1080.757,142.883,-70.270,174.497,22.868,153.879
C04176=1080.752,142.633,-70.250,174.494,22.866,153.879
C04177=1080.746,142.385,-70.230,174.492,22.864,153.879
C04178=1080.739,142.135,-70.208,174.490,22.862,153.878
C04179=1080.734,141.886,-70.187,174.488,22.859,153.878
C04180=1080.728,141.637,-70.167,174.486,22.857,153.878
C04181=1080.723,141.388,-70.147,174.484,22.855,153.878
C04182=1080.718,141.139,-70.126,174.482,22.853,153.878
C04183=1080.712,140.890,-70.106,174.481,22.851,153.878
C04184=1080.706,140.641,-70.086,174.478,22.849,153.878
C04185=1080.700,140.391,-70.065,174.476,22.847,153.877
C04186=1080.694,140.143,-70.045,174.475,22.845,153.877
C04187=1080.689,139.894,-70.024,174.472,22.842,153.877
C04188=1080.683,139.645,-70.004,174.470,22.840,153.877
C04189=1080.678,139.395,-69.985,174.468,22.838,153.877
C04190=1080.672,139.146,-69.965,174.466,22.836,153.877
C04191=1080.667,138.897,-69.944,174.465,22.834,153.876
C04192=1080.662,138.648,-69.923,174.463,22.831,153.876
C04193=1080.655,138.398,-69.903,174.460,22.829,153.876
C04194=1080.650,138.149,-69.883,174.459,22.827,153.876
C04195=1080.644,137.900,-69.863,174.457,22.825,153.876
C04196=1080.639,137.651,-69.842,174.454,22.823,153.876
C04197=1080.633,137.403,-69.822,174.453,22.821,153.875
C04198=1080.627,137.153,-69.802,174.450,22.818,153.875
C04199=1080.622,136.904,-69.782,174.449,22.817,153.875
C04200=1080.616,136.655,-69.762,174.447,22.814,153.875
C04201=1080.610,136.406,-69.742,174.444,22.812,153.875
C04202=1080.604,136.157,-69.722,174.443,22.810,153.875
C04203=1080.599,135.907,-69.701,174.441,22.808,153.875
C04204=1080.593,135.659,-69.681,174.439,22.806,153.874
C04205=1080.588,135.409,-69.661,174.437,22.804,153.874
C04206=1080.582,135.160,-69.641,174.435,22.801,153.874
C04207=1080.576,134.911,-69.621,174.433,22.799,153.874
C04208=1080.570,134.662,-69.601,174.431,22.797,153.874
C04209=1080.566,134.412,-69.581,174.429,22.794,153.874
C04210=1080.560,134.164,-69.561,174.427,22.793,153.873
C04211=1080.554,133.915,-69.541,174.425,22.790,153.873
C04212=1080.548,133.666,-69.520,174.424,22.788,153.873
C04213=1080.543,133.416,-69.501,174.421,22.786,153.873
C04214=1080.537,133.167,-69.481,174.420,22.784,153.873
C04215=1080.531,132.918,-69.461,174.418,22.781,153.872
C04216=1080.526,132.668,-69.441,174.415,22.779,153.872
C04217=1080.520,132.420,-69.421,174.414,22.777,153.872
C04218=1080.514,132.171,-69.401,174.412,22.775,153.872
C04219=1080.509,131.921,-69.381,174.410,22.773,153.872
C04220=1080.503,131.672,-69.361,174.408,22.771,153.872
C04221=1080.497,131.423,-69.341,174.406,22.768,153.872
C04222=1080.492,131.174,-69.322,174.404,22.767,153.871
C04223=1080.487,130.925,-69.301,174.402,22.764,153.871
C04224=1080.481,130.676,-69.281,174.400,22.762,153.871
C04225=1080.475,130.427,-69.262,174.398,22.760,153.871
C04226=1080.469,130.178,-69.242,174.396,22.758,153.871
C04227=1080.463,129.928,-69.223,174.394,22.756,153.871
C04228=1080.458,129.679,-69.202,174.392,22.753,153.870
C04229=1080.452,129.430,-69.182,174.391,22.751,153.870
C04230=1080.446,129.181,-69.163,174.388,22.749,153.870
C04231=1080.440,128.932,-69.143,174.387,22.747,153.870
C04232=1080.434,128.682,-69.124,174.385,22.745,153.870
C04233=1080.428,128.433,-69.104,174.382,22.743,153.870
C04234=1080.423,128.184,-69.084,174.381,22.741,153.869
C04235=1080.418,127.935,-69.064,174.379,22.738,153.869
C04236=1080.411,127.655,-69.042,174.377,22.736,153.869
C04237=1080.405,127.375,-69.020,174.375,22.734,153.869
C04238=1080.398,127.094,-68.997,174.373,22.731,153.869
C04239=1080.391,126.815,-68.976,174.371,22.729,153.869
C04240=1080.386,126.565,-68.956,174.368,22.726,153.868
C04241=1080.381,126.315,-68.937,174.367,22.724,153.868
C04242=1080.375,126.067,-68.917,174.365,22.722,153.868
C04243=1080.369,125.817,-68.898,174.363,22.720,153.868
C04244=1080.363,125.568,-68.878,174.361,22.718,153.868
C04245=1080.357,125.319,-68.858,174.359,22.715,153.867
C04246=1080.351,125.070,-68.838,174.357,22.713,153.867
C04247=1080.346,124.820,-68.819,174.355,22.711,153.867
C04248=1080.341,124.571,-68.799,174.354,22.709,153.867
C04249=1080.335,124.322,-68.779,174.351,22.707,153.867
C04250=1080.329,124.073,-68.760,174.350,22.705,153.867
C04251=1080.324,123.824,-68.741,174.348,22.702,153.866
C04252=1080.318,123.575,-68.721,174.346,22.700,153.866
C04253=1080.312,123.326,-68.702,174.344,22.698,153.866
C04254=1080.306,123.076,-68.683,174.343,22.696,153.866
C04255=1080.300,122.827,-68.663,174.340,22.694,153.866
C04256=1080.295,122.578,-68.644,174.338,22.691,153.866
C04257=1080.290,122.328,-68.624,174.337,22.689,153.865
C04258=1080.284,122.079,-68.604,174.334,22.687,153.865
C04259=1080.279,121.831,-68.585,174.333,22.685,153.865
C04260=1080.273,121.581,-68.566,174.331,22.682,153.865
C04261=1080.267,121.332,-68.546,174.329,22.680,153.865
C04262=1080.261,121.083,-68.526,174.327,22.678,153.865
C04263=1080.256,120.834,-68.507,174.326,22.676,153.864
C04264=1080.250,120.584,-68.488,174.324,22.673,153.864
C04265=1080.245,120.336,-68.468,174.322,22.671,153.864
C04266=1080.239,120.087,-68.449,174.320,22.669,153.864
C04267=1080.233,119.837,-68.430,174.318,22.667,153.864
C04268=1080.228,119.588,-68.411,174.316,22.664,153.863
C04269=1080.222,119.338,-68.391,174.315,22.662,153.863
C04270=1080.216,119.089,-68.371,174.313,22.660,153.863
C04271=1080.211,118.841,-68.353,174.311,22.658,153.863
C04272=1080.205,118.591,-68.333,174.309,22.655,153.863
C04273=1080.199,118.342,-68.314,174.307,22.653,153.862
C04274=1080.194,118.092,-68.294,174.305,22.651,153.862
C04275=1080.189,117.843,-68.275,174.303,22.648,153.862
C04276=1080.183,117.595,-68.255,174.302,22.647,153.862
C04277=1080.178,117.345,-68.236,174.299,22.644,153.862
C04278=1080.172,117.096,-68.217,174.298,22.642,153.861
C04279=1080.167,116.847,-68.198,174.296,22.640,153.861
C04280=1080.161,116.598,-68.179,174.295,22.638,153.861
C04281=1080.156,116.348,-68.160,174.292,22.635,153.861
C04282=1080.150,116.099,-68.140,174.291,22.633,153.861
C04283=1080.145,115.850,-68.121,174.289,22.631,153.861
C04284=1080.139,115.601,-68.102,174.287,22.628,153.860
C04285=1080.133,115.351,-68.083,174.285,22.626,153.860
C04286=1080.128,115.102,-68.064,174.284,22.624,153.860
C04287=1080.123,114.853,-68.045,174.282,22.621,153.860
C04288=1080.117,114.604,-68.026,174.280,22.619,153.859
C04289=1080.111,114.354,-68.006,174.278,22.616,153.859
C04290=1080.105,114.105,-67.988,174.277,22.615,153.859
C04291=1080.100,113.856,-67.969,174.274,22.612,153.859
C04292=1080.094,113.607,-67.950,174.273,22.610,153.859
C04293=1080.088,113.357,-67.930,174.271,22.608,153.858
C04294=1080.083,113.108,-67.911,174.269,22.606,153.858
C04295=1080.077,112.860,-67.893,174.267,22.603,153.858
C04296=1080.071,112.610,-67.874,174.266,22.601,153.858
C04297=1080.065,112.361,-67.854,174.264,22.599,153.858
C04298=1080.060,112.112,-67.835,174.262,22.597,153.858
C04299=1080.055,111.862,-67.816,174.260,22.594,153.857
C04300=1080.048,111.582,-67.795,174.259,22.592,153.857
C04301=1080.041,111.302,-67.774,174.256,22.589,153.857
C04302=1080.035,111.021,-67.752,174.254,22.587,153.857
C04303=1080.028,110.741,-67.731,174.252,22.584,153.856
C04304=1080.023,110.492,-67.712,174.251,22.582,153.856
C04305=1080.018,110.243,-67.693,174.248,22.580,153.856
C04306=1080.011,109.994,-67.675,174.247,22.578,153.856
C04307=1080.005,109.744,-67.655,174.245,22.575,153.856
C04308=1080.000,109.496,-67.637,174.243,22.573,153.856
C04309=1079.994,109.246,-67.619,174.241,22.571,153.855
C04310=1079.989,108.996,-67.599,174.240,22.569,153.855
C04311=1079.983,108.747,-67.580,174.238,22.566,153.855
C04312=1079.977,108.499,-67.562,174.236,22.564,153.855
C04313=1079.971,108.249,-67.543,174.234,22.562,153.855
C04314=1079.965,107.999,-67.525,174.233,22.560,153.854
C04315=1079.960,107.751,-67.506,174.230,22.557,153.854
C04316=1079.954,107.501,-67.487,174.229,22.555,153.854
C04317=1079.948,107.252,-67.468,174.227,22.553,153.854
C04318=1079.943,107.003,-67.450,174.225,22.551,153.854
C04319=1079.938,106.753,-67.431,174.224,22.548,153.853
C04320=1079.931,106.504,-67.412,174.222,22.546,153.853
C04321=1079.926,106.255,-67.393,174.221,22.544,153.853
C04322=1079.920,106.006,-67.375,174.218,22.541,153.853
C04323=1079.914,105.756,-67.356,174.217,22.539,153.853
C04324=1079.909,105.508,-67.337,174.215,22.537,153.852
C04325=1079.903,105.258,-67.318,174.213,22.535,153.852
C04326=1079.898,105.009,-67.300,174.211,22.532,153.852
C04327=1079.892,104.760,-67.282,174.210,22.530,153.852
C04328=1079.886,104.511,-67.262,174.208,22.528,153.852
C04329=1079.881,104.261,-67.244,174.206,22.525,153.851
C04330=1079.875,104.012,-67.225,174.204,22.523,153.851
C04331=1079.870,103.763,-67.207,174.203,22.521,153.851
C04332=1079.863,103.514,-67.189,174.201,22.519,153.851
C04333=1079.858,103.264,-67.169,174.199,22.516,153.851
C04334=1079.853,103.015,-67.151,174.198,22.514,153.850
C04335=1079.847,102.766,-67.133,174.196,22.512,153.850
C04336=1079.841,102.517,-67.114,174.194,22.509,153.850
C04337=1079.835,102.267,-67.096,174.192,22.507,153.850
C04338=1079.830,102.018,-67.077,174.191,22.505,153.850
C04339=1079.824,101.769,-67.059,174.189,22.502,153.849
C04340=1079.818,101.519,-67.040,174.187,22.500,153.849
C04341=1079.813,101.270,-67.022,174.185,22.497,153.849
C04342=1079.807,101.021,-67.003,174.184,22.496,153.849
C04343=1079.802,100.772,-66.985,174.182,22.494,153.848
C04344=1079.796,100.522,-66.966,174.180,22.491,153.848
C04345=1079.790,100.273,-66.948,174.179,22.489,153.848
C04346=1079.784,100.024,-66.930,174.177,22.486,153.848
C04347=1079.779,99.774,-66.911,174.175,22.484,153.848
C04348=1079.773,99.526,-66.893,174.173,22.482,153.847
C04349=1079.768,99.276,-66.875,174.172,22.480,153.847
C04350=1079.762,99.027,-66.856,174.170,22.478,153.847
C04351=1079.756,98.778,-66.838,174.168,22.475,153.847
C04352=1079.750,98.528,-66.819,174.167,22.473,153.847
C04353=1079.744,98.279,-66.802,174.164,22.471,153.846
C04354=1079.738,98.030,-66.783,174.163,22.468,153.846
C04355=1079.733,97.781,-66.765,174.161,22.466,153.846
C04356=1079.727,97.531,-66.746,174.160,22.463,153.846
C04357=1079.721,97.282,-66.728,174.157,22.461,153.846
C04358=1079.716,97.032,-66.710,174.156,22.459,153.845
C04359=1079.710,96.784,-66.692,174.155,22.457,153.845
C04360=1079.704,96.534,-66.674,174.152,22.454,153.845
C04361=1079.699,96.285,-66.656,174.151,22.452,153.845
C04362=1079.693,96.036,-66.637,174.149,22.450,153.845
C04363=1079.687,95.787,-66.619,174.148,22.447,153.844
C04364=1079.681,95.506,-66.599,174.145,22.445,153.844
C04365=1079.674,95.226,-66.578,174.143,22.442,153.844
C04366=1079.668,94.945,-66.558,174.142,22.440,153.844
C04367=1079.661,94.665,-66.537,174.140,22.437,153.843
C04368=1079.656,94.416,-66.520,174.139,22.435,153.843
C04369=1079.650,94.167,-66.500,174.136,22.432,153.843
C04370=1079.645,93.918,-66.483,174.135,22.430,153.843
C04371=1079.639,93.668,-66.465,174.133,22.427,153.842
C04372=1079.633,93.419,-66.446,174.132,22.426,153.842
C04373=1079.628,93.170,-66.428,174.130,22.423,153.842
C04374=1079.622,92.920,-66.410,174.128,22.421,153.842
C04375=1079.616,92.671,-66.393,174.127,22.418,153.842
C04376=1079.611,92.422,-66.374,174.125,22.416,153.841
C04377=1079.605,92.173,-66.356,174.123,22.414,153.841
C04378=1079.599,91.923,-66.338,174.121,22.411,153.841
C04379=1079.594,91.674,-66.320,174.120,22.409,153.841
C04380=1079.589,91.425,-66.302,174.118,22.407,153.840
C04381=1079.582,91.176,-66.284,174.116,22.404,153.840
C04382=1079.577,90.926,-66.266,174.115,22.402,153.840
C04383=1079.571,90.677,-66.248,174.113,22.399,153.840
C04384=1079.565,90.428,-66.231,174.111,22.398,153.840
C04385=1079.560,90.178,-66.212,174.110,22.395,153.839
C04386=1079.554,89.929,-66.195,174.108,22.393,153.839
C04387=1079.548,89.679,-66.176,174.106,22.391,153.839
C04388=1079.542,89.430,-66.158,174.104,22.388,153.839
C04389=1079.537,89.181,-66.141,174.103,22.386,153.839
C04390=1079.531,88.932,-66.123,174.102,22.384,153.838
C04391=1079.525,88.683,-66.105,174.099,22.381,153.838
C04392=1079.519,88.433,-66.087,174.098,22.379,153.838
C04393=1079.513,88.184,-66.070,174.096,22.377,153.838
C04394=1079.507,87.934,-66.052,174.095,22.374,153.837
C04395=1079.501,87.686,-66.034,174.093,22.372,153.837
C04396=1079.496,87.437,-66.016,174.091,22.369,153.837
C04397=1079.490,87.187,-65.998,174.090,22.368,153.837
C04398=1079.484,86.938,-65.980,174.088,22.365,153.837
C04399=1079.478,86.688,-65.963,174.086,22.363,153.836
C04400=1079.473,86.439,-65.945,174.085,22.360,153.836
C04401=1079.467,86.190,-65.927,174.083,22.358,153.836
C04402=1079.461,85.940,-65.909,174.082,22.356,153.836
C04403=1079.455,85.691,-65.892,174.080,22.354,153.835
C04404=1079.451,85.442,-65.874,174.078,22.351,153.835
C04405=1079.445,85.192,-65.856,174.077,22.349,153.835
C04406=1079.439,84.943,-65.838,174.075,22.346,153.835
C04407=1079.433,84.693,-65.820,174.073,22.344,153.835
C04408=1079.427,84.444,-65.803,174.072,22.342,153.834
C04409=1079.422,84.195,-65.785,174.070,22.340,153.834
C04410=1079.416,83.946,-65.767,174.068,22.337,153.834
C04411=1079.410,83.697,-65.750,174.066,22.335,153.834
C04412=1079.405,83.447,-65.732,174.065,22.332,153.833
C04413=1079.399,83.197,-65.715,174.064,22.330,153.833
C04414=1079.393,82.948,-65.697,174.061,22.328,153.833
C04415=1079.388,82.699,-65.680,174.060,22.325,153.833
C04416=1079.382,82.449,-65.662,174.059,22.323,153.833
C04417=1079.376,82.201,-65.645,174.057,22.320,153.832
C04418=1079.370,81.952,-65.627,174.055,22.319,153.832
C04419=1079.364,81.702,-65.610,174.053,22.316,153.832
C04420=1079.358,81.453,-65.592,174.052,22.313,153.832
C04421=1079.353,81.204,-65.574,174.051,22.311,153.831
C04422=1079.348,80.954,-65.557,174.049,22.308,153.831
C04423=1079.341,80.704,-65.539,174.047,22.307,153.831
C04424=1079.336,80.455,-65.522,174.046,22.304,153.831
C04425=1079.330,80.206,-65.504,174.044,22.301,153.830
C04426=1079.325,79.957,-65.487,174.042,22.299,153.830
C04427=1079.319,79.707,-65.470,174.040,22.297,153.830
C04428=1079.313,79.427,-65.449,174.039,22.294,153.830
C04429=1079.306,79.147,-65.430,174.037,22.291,153.829
C04430=1079.300,78.867,-65.411,174.035,22.288,153.829
C04431=1079.294,78.586,-65.391,174.034,22.286,153.829
C04432=1079.288,78.337,-65.373,174.031,22.284,153.829
C04433=1079.282,78.088,-65.356,174.030,22.281,153.828
C04434=1079.277,77.839,-65.339,174.029,22.279,153.828
C04435=1079.271,77.589,-65.321,174.027,22.276,153.828
C04436=1079.265,77.340,-65.304,174.025,22.275,153.828
C04437=1079.259,77.091,-65.286,174.024,22.272,153.828
C04438=1079.254,76.841,-65.270,174.022,22.270,153.827
C04439=1079.247,76.592,-65.252,174.021,22.267,153.827
C04440=1079.242,76.343,-65.234,174.019,22.265,153.827
C04441=1079.237,76.093,-65.218,174.017,22.263,153.827
C04442=1079.230,75.844,-65.201,174.016,22.260,153.826
C04443=1079.224,75.594,-65.183,174.014,22.258,153.826
C04444=1079.219,75.345,-65.166,174.012,22.255,153.826
C04445=1079.214,75.096,-65.148,174.011,22.253,153.826
C04446=1079.207,74.847,-65.131,174.009,22.251,153.826
C04447=1079.201,74.597,-65.114,174.008,22.248,153.825
C04448=1079.196,74.348,-65.096,174.006,22.246,153.825
C04449=1079.191,74.098,-65.080,174.004,22.243,153.825
C04450=1079.185,73.849,-65.063,174.003,22.242,153.825
C04451=1079.179,73.600,-65.045,174.002,22.239,153.824
C04452=1079.173,73.350,-65.028,174.000,22.236,153.824
C04453=1079.167,73.101,-65.011,173.998,22.234,153.824
C04454=1079.162,72.851,-64.994,173.997,22.232,153.824
C04455=1079.156,72.602,-64.976,173.995,22.229,153.823
C04456=1079.150,72.354,-64.959,173.994,22.227,153.823
C04457=1079.144,72.103,-64.942,173.992,22.225,153.823
C04458=1079.139,71.854,-64.925,173.990,22.222,153.823
C04459=1079.133,71.605,-64.908,173.989,22.220,153.822
C04460=1079.127,71.356,-64.891,173.988,22.217,153.822
C04461=1079.122,71.106,-64.874,173.985,22.215,153.822
C04462=1079.116,70.857,-64.857,173.984,22.213,153.822
C04463=1079.110,70.607,-64.840,173.983,22.210,153.821
C04464=1079.104,70.358,-64.822,173.981,22.208,153.821
C04465=1079.098,70.109,-64.806,173.979,22.205,153.821
C04466=1079.093,69.860,-64.788,173.978,22.203,153.821
C04467=1079.088,69.610,-64.772,173.976,22.201,153.821
C04468=1079.081,69.361,-64.755,173.975,22.198,153.820
C04469=1079.076,69.111,-64.737,173.973,22.196,153.820
C04470=1079.069,68.862,-64.720,173.971,22.194,153.820
C04471=1079.064,68.613,-64.704,173.970,22.191,153.820
C04472=1079.058,68.363,-64.687,173.969,22.189,153.819
C04473=1079.053,68.114,-64.670,173.967,22.186,153.819
C04474=1079.047,67.865,-64.653,173.965,22.184,153.819
C04475=1079.041,67.616,-64.636,173.964,22.182,153.819
C04476=1079.035,67.365,-64.619,173.962,22.179,153.818
C04477=1079.029,67.116,-64.602,173.961,22.177,153.818
C04478=1079.024,66.867,-64.585,173.959,22.175,153.818
C04479=1079.018,66.618,-64.569,173.957,22.172,153.818
C04480=1079.013,66.368,-64.552,173.956,22.170,153.817
C04481=1079.006,66.119,-64.535,173.955,22.168,153.817
C04482=1079.001,65.870,-64.518,173.953,22.165,153.817
C04483=1078.995,65.621,-64.501,173.951,22.163,153.817
C04484=1078.990,65.371,-64.484,173.950,22.160,153.816
C04485=1078.983,65.121,-64.468,173.948,22.157,153.816
C04486=1078.978,64.872,-64.451,173.947,22.156,153.816
C04487=1078.972,64.623,-64.434,173.945,22.153,153.816
C04488=1078.966,64.373,-64.417,173.943,22.151,153.816
C04489=1078.961,64.124,-64.401,173.942,22.148,153.815
C04490=1078.954,63.875,-64.384,173.941,22.146,153.815
C04491=1078.948,63.626,-64.367,173.938,22.144,153.815
C04492=1078.942,63.345,-64.349,173.937,22.141,153.815
C04493=1078.935,63.065,-64.330,173.935,22.138,153.814
C04494=1078.929,62.785,-64.310,173.933,22.135,153.814
C04495=1078.922,62.504,-64.292,173.932,22.133,153.814
C04496=1078.916,62.254,-64.276,173.930,22.131,153.814
C04497=1078.910,62.006,-64.259,173.928,22.128,153.813
C04498=1078.904,61.756,-64.242,173.927,22.126,153.813
C04499=1078.898,61.507,-64.226,173.926,22.124,153.813
C04500=1078.893,61.257,-64.209,173.924,22.121,153.813
C04501=1078.887,61.008,-64.193,173.922,22.119,153.812
C04502=1078.881,60.758,-64.177,173.921,22.117,153.812
C04503=1078.875,60.510,-64.160,173.919,22.114,153.812
C04504=1078.869,60.259,-64.142,173.918,22.112,153.812
C04505=1078.863,60.010,-64.126,173.916,22.109,153.811
C04506=1078.857,59.761,-64.110,173.914,22.107,153.811
C04507=1078.851,59.511,-64.094,173.913,22.105,153.811
C04508=1078.846,59.262,-64.077,173.912,22.102,153.811
C04509=1078.840,59.012,-64.061,173.910,22.100,153.810
C04510=1078.834,58.764,-64.044,173.908,22.097,153.810
C04511=1078.828,58.514,-64.027,173.907,22.095,153.810
C04512=1078.823,58.265,-64.011,173.906,22.093,153.810
C04513=1078.817,58.015,-63.994,173.904,22.090,153.810
C04514=1078.811,57.766,-63.978,173.902,22.088,153.809
C04515=1078.805,57.517,-63.962,173.901,22.086,153.809
C04516=1078.800,57.267,-63.945,173.899,22.083,153.809
C04517=1078.794,57.018,-63.929,173.898,22.081,153.809
C04518=1078.788,56.768,-63.912,173.896,22.078,153.808
C04519=1078.782,56.519,-63.896,173.894,22.076,153.808
C04520=1078.776,56.270,-63.880,173.893,22.074,153.808
C04521=1078.770,56.020,-63.863,173.892,22.071,153.808
C04522=1078.765,55.771,-63.847,173.891,22.069,153.807
C04523=1078.759,55.521,-63.831,173.888,22.066,153.807
C04524=1078.753,55.272,-63.814,173.887,22.064,153.807
C04525=1078.747,55.022,-63.798,173.886,22.062,153.807
C04526=1078.741,54.773,-63.781,173.884,22.059,153.806
C04527=1078.736,54.523,-63.765,173.882,22.057,153.806
C04528=1078.730,54.274,-63.749,173.881,22.054,153.806
C04529=1078.724,54.025,-63.732,173.880,22.052,153.806
C04530=1078.718,53.775,-63.716,173.878,22.050,153.805
C04531=1078.712,53.526,-63.700,173.877,22.047,153.805
C04532=1078.707,53.276,-63.683,173.875,22.045,153.805
C04533=1078.701,53.027,-63.667,173.873,22.042,153.805
C04534=1078.695,52.778,-63.650,173.872,22.040,153.804
C04535=1078.689,52.528,-63.634,173.871,22.037,153.804
C04536=1078.683,52.280,-63.618,173.869,22.035,153.804
C04537=1078.678,52.030,-63.603,173.867,22.033,153.804
C04538=1078.672,51.780,-63.587,173.866,22.030,153.803
C04539=1078.666,51.531,-63.570,173.865,22.028,153.803
C04540=1078.661,51.281,-63.553,173.863,22.025,153.803
C04541=1078.655,51.032,-63.537,173.861,22.023,153.803
C04542=1078.649,50.783,-63.521,173.860,22.020,153.802
C04543=1078.643,50.533,-63.505,173.858,22.018,153.802
C04544=1078.637,50.283,-63.489,173.857,22.016,153.802
C04545=1078.631,50.034,-63.473,173.856,22.013,153.802
C04546=1078.626,49.785,-63.456,173.854,22.011,153.801
C04547=1078.621,49.536,-63.440,173.852,22.008,153.801
C04548=1078.615,49.286,-63.424,173.851,22.006,153.801
C04549=1078.609,49.037,-63.408,173.850,22.004,153.801
C04550=1078.603,48.787,-63.392,173.848,22.001,153.800
C04551=1078.597,48.538,-63.376,173.846,21.999,153.800
C04552=1078.591,48.288,-63.360,173.845,21.996,153.800
C04553=1078.586,48.040,-63.344,173.844,21.994,153.800
C04554=1078.580,47.790,-63.328,173.842,21.991,153.799
C04555=1078.575,47.540,-63.311,173.841,21.989,153.799
C04556=1078.568,47.260,-63.294,173.839,21.986,153.799
C04557=1078.562,46.979,-63.275,173.837,21.983,153.798
C04558=1078.555,46.699,-63.257,173.835,21.980,153.798
C04559=1078.549,46.418,-63.239,173.834,21.978,153.798
C04560=1078.544,46.169,-63.223,173.833,21.975,153.798
C04561=1078.538,45.919,-63.207,173.831,21.973,153.797
C04562=1078.532,45.670,-63.191,173.830,21.971,153.797
C04563=1078.526,45.420,-63.175,173.828,21.968,153.797
C04564=1078.520,45.171,-63.159,173.826,21.965,153.797
C04565=1078.515,44.922,-63.143,173.825,21.963,153.796
C04566=1078.509,44.672,-63.128,173.824,21.961,153.796
C04567=1078.503,44.423,-63.111,173.823,21.958,153.796
C04568=1078.498,44.173,-63.095,173.821,21.956,153.796
C04569=1078.493,43.924,-63.079,173.819,21.953,153.795
C04570=1078.487,43.675,-63.063,173.818,21.951,153.795
C04571=1078.480,43.425,-63.048,173.816,21.948,153.795
C04572=1078.475,43.176,-63.032,173.815,21.946,153.795
C04573=1078.469,42.926,-63.016,173.814,21.943,153.794
C04574=1078.464,42.677,-63.001,173.812,21.941,153.794
C04575=1078.458,42.428,-62.984,173.810,21.939,153.794
C04576=1078.452,42.178,-62.969,173.809,21.936,153.794
C04577=1078.446,41.928,-62.953,173.808,21.934,153.793
C04578=1078.440,41.678,-62.937,173.806,21.932,153.793
C04579=1078.434,41.430,-62.922,173.804,21.929,153.793
C04580=1078.428,41.181,-62.905,173.803,21.926,153.793
C04581=1078.423,40.931,-62.890,173.802,21.924,153.792
C04582=1078.417,40.681,-62.874,173.801,21.922,153.792
C04583=1078.411,40.431,-62.858,173.798,21.919,153.792
C04584=1078.406,40.183,-62.842,173.797,21.917,153.792
C04585=1078.400,39.933,-62.827,173.796,21.915,153.791
C04586=1078.393,39.684,-62.811,173.795,21.912,153.791
C04587=1078.388,39.434,-62.795,173.793,21.909,153.791
C04588=1078.382,39.185,-62.780,173.791,21.907,153.790
C04589=1078.377,38.935,-62.764,173.790,21.905,153.790
C04590=1078.371,38.686,-62.748,173.788,21.902,153.790
C04591=1078.366,38.436,-62.733,173.787,21.900,153.790
C04592=1078.359,38.187,-62.718,173.786,21.897,153.789
C04593=1078.353,37.937,-62.701,173.784,21.895,153.789
C04594=1078.348,37.687,-62.686,173.782,21.892,153.789
C04595=1078.342,37.439,-62.670,173.781,21.890,153.789
C04596=1078.336,37.189,-62.655,173.780,21.887,153.788
C04597=1078.330,36.940,-62.639,173.779,21.886,153.788
C04598=1078.324,36.690,-62.623,173.776,21.883,153.788
C04599=1078.318,36.440,-62.608,173.775,21.880,153.788
C04600=1078.313,36.192,-62.592,173.774,21.878,153.788
C04601=1078.307,35.942,-62.577,173.773,21.876,153.787
C04602=1078.301,35.692,-62.562,173.771,21.873,153.787
C04603=1078.295,35.443,-62.546,173.769,21.871,153.787
C04604=1078.290,35.193,-62.530,173.768,21.869,153.787
C04605=1078.283,34.944,-62.515,173.767,21.866,153.786
C04606=1078.277,34.694,-62.499,173.765,21.864,153.786
C04607=1078.272,34.445,-62.485,173.763,21.861,153.786
C04608=1078.266,34.196,-62.468,173.762,21.859,153.786
C04609=1078.260,33.946,-62.453,173.761,21.856,153.785
C04610=1078.254,33.697,-62.438,173.759,21.854,153.785
C04611=1078.249,33.447,-62.423,173.758,21.852,153.785
C04612=1078.243,33.198,-62.407,173.757,21.849,153.784
C04613=1078.236,32.948,-62.392,173.755,21.847,153.784
C04614=1078.231,32.699,-62.376,173.753,21.844,153.784
C04615=1078.224,32.450,-62.361,173.752,21.842,153.784
C04616=1078.219,32.200,-62.345,173.751,21.839,153.783
C04617=1078.214,31.951,-62.330,173.749,21.837,153.783
C04618=1078.207,31.701,-62.315,173.747,21.835,153.783
C04619=1078.201,31.452,-62.299,173.746,21.832,153.783
C04620=1078.196,31.171,-62.282,173.745,21.830,153.782
C04621=1078.189,30.891,-62.265,173.743,21.827,153.782
C04622=1078.183,30.610,-62.248,173.742,21.824,153.782
C04623=1078.176,30.330,-62.230,173.740,21.821,153.782
C04624=1078.170,30.080,-62.215,173.738,21.819,153.781
C04625=1078.164,29.831,-62.200,173.737,21.816,153.781
C04626=1078.159,29.581,-62.185,173.735,21.814,153.781
C04627=1078.152,29.331,-62.170,173.734,21.812,153.781
C04628=1078.147,29.083,-62.154,173.733,21.809,153.780
C04629=1078.141,28.833,-62.139,173.732,21.807,153.780
C04630=1078.135,28.583,-62.123,173.729,21.804,153.780
C04631=1078.129,28.334,-62.109,173.728,21.802,153.780
C04632=1078.124,28.084,-62.093,173.727,21.799,153.779
C04633=1078.118,27.835,-62.079,173.726,21.797,153.779
C04634=1078.112,27.585,-62.063,173.724,21.795,153.779
C04635=1078.105,27.336,-62.047,173.722,21.792,153.779
C04636=1078.100,27.087,-62.032,173.721,21.790,153.778
C04637=1078.094,26.837,-62.017,173.720,21.788,153.778
C04638=1078.088,26.587,-62.002,173.719,21.785,153.778
C04639=1078.083,26.338,-61.987,173.716,21.783,153.778
C04640=1078.076,26.089,-61.972,173.715,21.780,153.777
C04641=1078.071,25.839,-61.957,173.714,21.778,153.777
C04642=1078.065,25.590,-61.942,173.713,21.776,153.777
C04643=1078.059,25.340,-61.927,173.711,21.773,153.777
C04644=1078.053,25.091,-61.912,173.709,21.771,153.776
C04645=1078.047,24.841,-61.897,173.708,21.768,153.776
C04646=1078.042,24.592,-61.882,173.707,21.766,153.776
C04647=1078.035,24.342,-61.867,173.705,21.763,153.776
C04648=1078.030,24.092,-61.851,173.704,21.761,153.775
C04649=1078.024,23.843,-61.837,173.702,21.759,153.775
C04650=1078.018,23.593,-61.822,173.701,21.756,153.775
C04651=1078.013,23.344,-61.807,173.700,21.754,153.775
C04652=1078.006,23.095,-61.792,173.698,21.752,153.775
C04653=1078.000,22.846,-61.777,173.697,21.749,153.774
C04654=1077.995,22.596,-61.762,173.695,21.747,153.774
C04655=1077.988,22.346,-61.747,173.694,21.744,153.774
C04656=1077.983,22.097,-61.731,173.692,21.742,153.773
C04657=1077.977,21.847,-61.717,173.691,21.739,153.773
C04658=1077.971,21.598,-61.702,173.690,21.737,153.773
C04659=1077.966,21.348,-61.686,173.688,21.735,153.773
C04660=1077.960,21.099,-61.672,173.687,21.733,153.772
C04661=1077.954,20.849,-61.658,173.685,21.730,153.772
C04662=1077.949,20.600,-61.642,173.684,21.728,153.772
C04663=1077.942,20.350,-61.627,173.683,21.725,153.772
C04664=1077.937,20.101,-61.613,173.681,21.723,153.771
C04665=1077.931,19.851,-61.597,173.679,21.720,153.771
C04666=1077.925,19.602,-61.583,173.678,21.718,153.771
C04667=1077.919,19.352,-61.568,173.677,21.715,153.771
C04668=1077.913,19.104,-61.553,173.676,21.713,153.770
C04669=1077.908,18.853,-61.538,173.674,21.711,153.770
C04670=1077.902,18.604,-61.524,173.672,21.708,153.770
C04671=1077.895,18.354,-61.509,173.671,21.706,153.770
C04672=1077.890,18.105,-61.494,173.670,21.704,153.770
C04673=1077.883,17.856,-61.479,173.668,21.701,153.769
C04674=1077.878,17.606,-61.464,173.667,21.699,153.769
C04675=1077.872,17.356,-61.450,173.665,21.696,153.769
C04676=1077.866,17.107,-61.435,173.664,21.694,153.768
C04677=1077.860,16.858,-61.420,173.663,21.691,153.768
C04678=1077.855,16.608,-61.405,173.661,21.690,153.768
C04679=1077.849,16.358,-61.391,173.659,21.687,153.768
C04680=1077.843,16.109,-61.376,173.658,21.684,153.767
C04681=1077.837,15.859,-61.361,173.657,21.682,153.767
C04682=1077.831,15.610,-61.347,173.656,21.680,153.767
C04683=1077.826,15.360,-61.332,173.654,21.677,153.767
C04684=1077.819,15.081,-61.316,173.652,21.674,153.766
C04685=1077.812,14.802,-61.299,173.651,21.672,153.766
C04686=1077.806,14.522,-61.283,173.649,21.669,153.766
C04687=1077.799,14.244,-61.266,173.648,21.667,153.766
C04688=1077.793,13.994,-61.252,173.646,21.664,153.766
C04689=1077.787,13.745,-61.238,173.645,21.662,153.765
C04690=1077.781,13.495,-61.223,173.643,21.660,153.765
C04691=1077.776,13.246,-61.209,173.642,21.657,153.765
C04692=1077.769,12.996,-61.194,173.641,21.655,153.764
C04693=1077.763,12.747,-61.179,173.639,21.652,153.764
C04694=1077.757,12.497,-61.165,173.638,21.650,153.764
C04695=1077.752,12.248,-61.150,173.636,21.648,153.764
C04696=1077.746,11.999,-61.136,173.635,21.646,153.764
C04697=1077.740,11.749,-61.122,173.634,21.643,153.763
C04698=1077.734,11.500,-61.107,173.632,21.641,153.763
C04699=1077.728,11.249,-61.093,173.630,21.638,153.763
C04700=1077.722,11.000,-61.078,173.629,21.636,153.763
C04701=1077.716,10.751,-61.063,173.628,21.634,153.762
C04702=1077.710,10.501,-61.049,173.627,21.631,153.762
C04703=1077.704,10.251,-61.034,173.625,21.629,153.762
C04704=1077.698,10.002,-61.021,173.623,21.627,153.762
C04705=1077.693,9.753,-61.006,173.622,21.625,153.762
C04706=1077.686,9.503,-60.992,173.621,21.622,153.761
C04707=1077.681,9.254,-60.977,173.620,21.620,153.761
C04708=1077.674,9.004,-60.962,173.617,21.617,153.761
C04709=1077.669,8.754,-60.948,173.616,21.615,153.760
C04710=1077.662,8.505,-60.933,173.615,21.613,153.760
C04711=1077.656,8.256,-60.920,173.614,21.610,153.760
C04712=1077.650,8.007,-60.906,173.613,21.608,153.760
C04713=1077.644,7.756,-60.891,173.610,21.606,153.760
C04714=1077.639,7.507,-60.877,173.609,21.603,153.759
C04715=1077.633,7.258,-60.863,173.608,21.601,153.759
C04716=1077.627,7.008,-60.848,173.607,21.599,153.759
C04717=1077.621,6.759,-60.834,173.606,21.596,153.759
C04718=1077.615,6.509,-60.819,173.603,21.594,153.758
C04719=1077.609,6.259,-60.805,173.602,21.591,153.758
C04720=1077.604,6.010,-60.791,173.601,21.589,153.758
C04721=1077.598,5.760,-60.776,173.600,21.587,153.758
C04722=1077.592,5.510,-60.763,173.598,21.584,153.757
C04723=1077.586,5.262,-60.748,173.596,21.582,153.757
C04724=1077.580,5.011,-60.734,173.595,21.580,153.757
C04725=1077.574,4.762,-60.719,173.594,21.577,153.757
C04726=1077.568,4.513,-60.706,173.593,21.575,153.757
C04727=1077.562,4.263,-60.692,173.591,21.573,153.756
C04728=1077.556,4.014,-60.677,173.589,21.570,153.756
C04729=1077.551,3.764,-60.663,173.588,21.568,153.756
C04730=1077.545,3.514,-60.649,173.587,21.565,153.755
C04731=1077.539,3.265,-60.634,173.585,21.563,153.755
C04732=1077.534,3.015,-60.621,173.584,21.561,153.755
C04733=1077.528,2.766,-60.607,173.582,21.558,153.755
C04734=1077.522,2.516,-60.592,173.581,21.556,153.755
C04735=1077.516,2.267,-60.578,173.580,21.554,153.754
C04736=1077.510,2.017,-60.565,173.578,21.552,153.754
C04737=1077.504,1.768,-60.550,173.577,21.549,153.754
C04738=1077.498,1.518,-60.536,173.576,21.547,153.754
C04739=1077.493,1.269,-60.522,173.574,21.544,153.753
C04740=1077.487,1.020,-60.507,173.573,21.542,153.753
C04741=1077.481,0.769,-60.493,173.571,21.540,153.753
C04742=1077.475,0.520,-60.479,173.570,21.537,153.753
C04743=1077.469,0.271,-60.465,173.569,21.535,153.752
C04744=1077.463,0.022,-60.451,173.567,21.533,153.752
C04745=1077.457,-0.229,-60.437,173.566,21.530,153.752
C04746=1077.452,-0.478,-60.423,173.565,21.528,153.752
C04747=1077.446,-0.727,-60.409,173.563,21.526,153.752
C04748=1077.440,-1.005,-60.393,173.561,21.523,153.751
C04749=1077.433,-1.282,-60.378,173.560,21.520,153.751
C04750=1077.427,-1.559,-60.362,173.559,21.518,153.751
C04751=1077.421,-1.836,-60.347,173.557,21.515,153.750
C04752=1077.415,-2.086,-60.333,173.555,21.513,153.750
C04753=1077.409,-2.335,-60.318,173.554,21.510,153.750
C04754=1077.403,-2.585,-60.305,173.553,21.508,153.750
C04755=1077.397,-2.834,-60.291,173.551,21.506,153.750
C04756=1077.392,-3.084,-60.277,173.550,21.503,153.749
C04757=1077.386,-3.334,-60.263,173.549,21.501,153.749
C04758=1077.379,-3.583,-60.249,173.547,21.499,153.749
C04759=1077.374,-3.832,-60.235,173.546,21.497,153.749
C04760=1077.368,-4.082,-60.221,173.544,21.494,153.748
C04761=1077.361,-4.332,-60.208,173.543,21.492,153.748
C04762=1077.356,-4.581,-60.194,173.541,21.489,153.748
C04763=1077.350,-4.831,-60.181,173.540,21.487,153.748
C04764=1077.344,-5.080,-60.167,173.539,21.485,153.747
C04765=1077.338,-5.331,-60.153,173.537,21.483,153.747
C04766=1077.332,-5.580,-60.139,173.535,21.480,153.747
C04767=1077.326,-5.829,-60.125,173.534,21.478,153.747
C04768=1077.320,-6.078,-60.111,173.533,21.476,153.747
C04769=1077.314,-6.328,-60.097,173.532,21.474,153.746
C04770=1077.308,-6.578,-60.083,173.530,21.471,153.746
C04771=1077.302,-6.827,-60.070,173.529,21.469,153.746
C04772=1077.297,-7.077,-60.056,173.527,21.466,153.746
C04773=1077.290,-7.326,-60.043,173.526,21.464,153.746
C04774=1077.284,-7.576,-60.029,173.525,21.462,153.745
C04775=1077.278,-7.826,-60.015,173.523,21.460,153.745
C04776=1077.273,-8.075,-60.002,173.522,21.457,153.745
C04777=1077.266,-8.324,-59.988,173.520,21.455,153.745
C04778=1077.261,-8.574,-59.974,173.519,21.453,153.744
C04779=1077.255,-8.824,-59.960,173.517,21.451,153.744
C04780=1077.249,-9.073,-59.947,173.516,21.448,153.744
C04781=1077.243,-9.323,-59.933,173.515,21.446,153.744
C04782=1077.237,-9.572,-59.920,173.514,21.444,153.743
C04783=1077.231,-9.822,-59.906,173.511,21.441,153.743
C04784=1077.225,-10.071,-59.893,173.510,21.439,153.743
C04785=1077.219,-10.321,-59.878,173.509,21.437,153.743
C04786=1077.213,-10.571,-59.865,173.508,21.434,153.743
C04787=1077.207,-10.820,-59.851,173.506,21.432,153.742
C04788=1077.201,-11.070,-59.838,173.505,21.430,153.742
C04789=1077.196,-11.319,-59.824,173.503,21.428,153.742
C04790=1077.190,-11.569,-59.812,173.502,21.425,153.742
C04791=1077.184,-11.819,-59.798,173.501,21.423,153.742
C04792=1077.178,-12.068,-59.785,173.499,21.421,153.741
C04793=1077.172,-12.318,-59.770,173.498,21.419,153.741
C04794=1077.166,-12.567,-59.757,173.497,21.417,153.741
C04795=1077.160,-12.817,-59.743,173.495,21.414,153.741
C04796=1077.154,-13.066,-59.730,173.493,21.412,153.741
C04797=1077.149,-13.316,-59.716,173.492,21.409,153.740
C04798=1077.143,-13.566,-59.703,173.491,21.407,153.740
C04799=1077.137,-13.815,-59.690,173.490,21.405,153.740
C04800=1077.131,-14.065,-59.676,173.488,21.403,153.740
C04801=1077.126,-14.314,-59.662,173.486,21.400,153.739
C04802=1077.119,-14.563,-59.649,173.485,21.398,153.739
C04803=1077.114,-14.813,-59.635,173.484,21.396,153.739
C04804=1077.108,-15.063,-59.623,173.483,21.394,153.739
C04805=1077.102,-15.313,-59.609,173.481,21.391,153.738
C04806=1077.096,-15.562,-59.595,173.480,21.389,153.738
C04807=1077.090,-15.812,-59.582,173.478,21.387,153.738
C04808=1077.084,-16.061,-59.568,173.477,21.384,153.738
C04809=1077.078,-16.311,-59.556,173.475,21.382,153.738
C04810=1077.072,-16.560,-59.542,173.474,21.380,153.738
C04811=1077.066,-16.810,-59.529,173.473,21.378,153.737
C04812=1077.059,-17.085,-59.514,173.471,21.376,153.737
C04813=1077.053,-17.361,-59.500,173.469,21.373,153.737
C04814=1077.046,-17.637,-59.484,173.468,21.371,153.737
C04815=1077.040,-17.912,-59.470,173.466,21.368,153.736
C04816=1077.034,-18.162,-59.457,173.465,21.366,153.736
C04817=1077.027,-18.411,-59.444,173.464,21.364,153.736
C04818=1077.022,-18.661,-59.430,173.462,21.362,153.736
C04819=1077.016,-18.910,-59.417,173.461,21.359,153.735
C04820=1077.010,-19.160,-59.404,173.459,21.357,153.735
C04821=1077.004,-19.409,-59.390,173.458,21.355,153.735
C04822=1076.998,-19.659,-59.378,173.456,21.352,153.735
C04823=1076.992,-19.908,-59.364,173.455,21.351,153.735
C04824=1076.986,-20.158,-59.351,173.454,21.349,153.735
C04825=1076.981,-20.408,-59.338,173.453,21.346,153.734
C04826=1076.974,-20.658,-59.324,173.450,21.344,153.734
C04827=1076.968,-20.907,-59.311,173.449,21.341,153.734
C04828=1076.962,-21.157,-59.299,173.448,21.339,153.734
C04829=1076.956,-21.407,-59.285,173.447,21.337,153.734
C04830=1076.950,-21.656,-59.272,173.445,21.335,153.733
C04831=1076.944,-21.906,-59.259,173.444,21.333,153.733
C04832=1076.938,-22.155,-59.246,173.443,21.331,153.733
C04833=1076.933,-22.405,-59.232,173.441,21.328,153.733
C04834=1076.927,-22.654,-59.219,173.439,21.326,153.733
C04835=1076.921,-22.904,-59.207,173.438,21.324,153.732
C04836=1076.915,-23.154,-59.193,173.437,21.322,153.732
C04837=1076.909,-23.403,-59.181,173.435,21.320,153.732
C04838=1076.904,-23.652,-59.167,173.434,21.318,153.732
C04839=1076.898,-23.902,-59.154,173.432,21.315,153.732
C04840=1076.892,-24.151,-59.141,173.431,21.313,153.731
C04841=1076.885,-24.401,-59.128,173.429,21.311,153.731
C04842=1076.880,-24.651,-59.115,173.428,21.308,153.731
C04843=1076.874,-24.900,-59.102,173.427,21.306,153.731
C04844=1076.868,-25.150,-59.089,173.426,21.304,153.731
C04845=1076.862,-25.399,-59.076,173.424,21.302,153.730
C04846=1076.856,-25.649,-59.063,173.422,21.300,153.730
C04847=1076.851,-25.899,-59.050,173.421,21.298,153.730
C04848=1076.845,-26.149,-59.037,173.420,21.295,153.730
C04849=1076.838,-26.398,-59.024,173.418,21.293,153.730
C04850=1076.833,-26.648,-59.011,173.417,21.291,153.729
C04851=1076.827,-26.898,-58.999,173.416,21.289,153.729
C04852=1076.820,-27.147,-58.985,173.415,21.287,153.729
C04853=1076.814,-27.397,-58.973,173.412,21.284,153.729
C04854=1076.808,-27.646,-58.960,173.411,21.282,153.729
C04855=1076.802,-27.896,-58.947,173.410,21.280,153.728
C04856=1076.796,-28.145,-58.934,173.409,21.278,153.728
C04857=1076.790,-28.395,-58.921,173.407,21.276,153.728
C04858=1076.784,-28.645,-58.909,173.406,21.274,153.728
C04859=1076.779,-28.894,-58.896,173.405,21.272,153.728
C04860=1076.773,-29.143,-58.883,173.403,21.269,153.727
C04861=1076.767,-29.393,-58.870,173.401,21.267,153.727
C04862=1076.761,-29.643,-58.857,173.400,21.265,153.727
C04863=1076.755,-29.893,-58.845,173.399,21.263,153.727
C04864=1076.749,-30.142,-58.831,173.397,21.261,153.727
C04865=1076.743,-30.392,-58.819,173.396,21.259,153.727
C04866=1076.737,-30.642,-58.806,173.395,21.257,153.726
C04867=1076.731,-30.891,-58.793,173.392,21.254,153.726
C04868=1076.725,-31.141,-58.781,173.391,21.252,153.726
C04869=1076.719,-31.391,-58.768,173.390,21.250,153.726
C04870=1076.712,-31.640,-58.755,173.389,21.248,153.726
C04871=1076.707,-31.890,-58.742,173.387,21.246,153.725
C04872=1076.701,-32.139,-58.730,173.386,21.244,153.725
C04873=1076.695,-32.388,-58.717,173.385,21.242,153.725
C04874=1076.689,-32.638,-58.704,173.383,21.240,153.725
C04875=1076.683,-32.888,-58.692,173.381,21.237,153.725
C04876=1076.676,-33.163,-58.677,173.380,21.235,153.725
C04877=1076.670,-33.437,-58.664,173.379,21.233,153.724
C04878=1076.664,-33.712,-58.649,173.377,21.230,153.724
C04879=1076.657,-33.986,-58.635,173.375,21.228,153.724
C04880=1076.651,-34.236,-58.623,173.374,21.226,153.724
C04881=1076.645,-34.486,-58.610,173.373,21.224,153.724
C04882=1076.639,-34.736,-58.598,173.371,21.222,153.723
C04883=1076.633,-34.985,-58.585,173.369,21.220,153.723
C04884=1076.627,-35.235,-58.572,173.368,21.218,153.723
C04885=1076.621,-35.484,-58.560,173.367,21.216,153.723
C04886=1076.615,-35.734,-58.548,173.365,21.214,153.723
C04887=1076.610,-35.984,-58.535,173.364,21.212,153.723
C04888=1076.603,-36.233,-58.522,173.363,21.209,153.722
C04889=1076.597,-36.483,-58.509,173.361,21.207,153.722
C04890=1076.592,-36.732,-58.497,173.360,21.205,153.722
C04891=1076.586,-36.982,-58.485,173.358,21.203,153.722
C04892=1076.580,-37.232,-58.472,173.357,21.201,153.722
C04893=1076.574,-37.482,-58.460,173.355,21.199,153.722
C04894=1076.568,-37.731,-58.446,173.354,21.197,153.721
C04895=1076.562,-37.980,-58.435,173.353,21.195,153.721
C04896=1076.556,-38.230,-58.422,173.351,21.193,153.721
C04897=1076.550,-38.480,-58.410,173.350,21.191,153.721
C04898=1076.544,-38.730,-58.397,173.349,21.189,153.721
C04899=1076.538,-38.979,-58.384,173.346,21.186,153.721
C04900=1076.532,-39.228,-58.373,173.345,21.184,153.720
C04901=1076.527,-39.478,-58.360,173.344,21.182,153.720
C04902=1076.521,-39.728,-58.348,173.342,21.180,153.720
C04903=1076.515,-39.978,-58.335,173.341,21.178,153.720
C04904=1076.508,-40.227,-58.323,173.340,21.176,153.720
C04905=1076.502,-40.477,-58.310,173.338,21.174,153.720
C04906=1076.497,-40.726,-58.298,173.337,21.173,153.719
C04907=1076.491,-40.976,-58.285,173.335,21.170,153.719
C04908=1076.484,-41.225,-58.273,173.334,21.168,153.719
C04909=1076.478,-41.475,-58.261,173.332,21.166,153.719
C04910=1076.473,-41.724,-58.249,173.331,21.164,153.719
C04911=1076.466,-41.974,-58.237,173.330,21.162,153.719
C04912=1076.460,-42.224,-58.224,173.328,21.160,153.719
C04913=1076.454,-42.474,-58.211,173.327,21.158,153.718
C04914=1076.448,-42.723,-58.199,173.326,21.156,153.718
C04915=1076.442,-42.973,-58.187,173.324,21.154,153.718
C04916=1076.436,-43.222,-58.175,173.322,21.152,153.718
C04917=1076.430,-43.472,-58.163,173.321,21.150,153.718
C04918=1076.424,-43.722,-58.150,173.319,21.148,153.718
C04919=1076.419,-43.971,-58.138,173.318,21.146,153.717
C04920=1076.412,-44.221,-58.126,173.317,21.144,153.717
C04921=1076.406,-44.471,-58.114,173.315,21.142,153.717
C04922=1076.400,-44.721,-58.102,173.314,21.140,153.717
C04923=1076.394,-44.970,-58.090,173.313,21.138,153.717
C04924=1076.388,-45.220,-58.078,173.311,21.136,153.717
C04925=1076.383,-45.470,-58.065,173.309,21.134,153.717
C04926=1076.376,-45.719,-58.053,173.308,21.132,153.716
C04927=1076.371,-45.968,-58.041,173.306,21.130,153.716
C04928=1076.365,-46.218,-58.028,173.305,21.128,153.716
C04929=1076.358,-46.468,-58.016,173.304,21.126,153.716
C04930=1076.353,-46.717,-58.004,173.302,21.124,153.716
C04931=1076.347,-46.967,-57.992,173.301,21.122,153.716
C04932=1076.340,-47.217,-57.980,173.300,21.120,153.715
C04933=1076.335,-47.466,-57.968,173.298,21.118,153.715
C04934=1076.329,-47.716,-57.956,173.297,21.116,153.715
C04935=1076.323,-47.966,-57.944,173.295,21.114,153.715
C04936=1076.317,-48.215,-57.931,173.294,21.112,153.715
C04937=1076.311,-48.465,-57.920,173.292,21.110,153.715
C04938=1076.305,-48.715,-57.908,173.291,21.108,153.714
C04939=1076.300,-48.964,-57.895,173.290,21.106,153.714
C04940=1076.293,-49.240,-57.882,173.288,21.104,153.714
C04941=1076.287,-49.514,-57.869,173.286,21.102,153.714
C04942=1076.279,-49.789,-57.856,173.285,21.100,153.714
C04943=1076.273,-50.065,-57.842,173.283,21.098,153.714
C04944=1076.267,-50.314,-57.830,173.282,21.096,153.714
C04945=1076.261,-50.564,-57.819,173.281,21.094,153.713
C04946=1076.255,-50.814,-57.806,173.278,21.091,153.713
C04947=1076.249,-51.063,-57.795,173.277,21.089,153.713
C04948=1076.243,-51.313,-57.782,173.276,21.088,153.713
C04949=1076.237,-51.563,-57.771,173.274,21.086,153.713
C04950=1076.230,-51.812,-57.759,173.273,21.084,153.713
C04951=1076.225,-52.062,-57.747,173.272,21.082,153.713
C04952=1076.218,-52.311,-57.735,173.270,21.080,153.713
C04953=1076.212,-52.561,-57.724,173.269,21.079,153.712
C04954=1076.206,-52.810,-57.711,173.267,21.077,153.712
C04955=1076.200,-53.060,-57.699,173.266,21.075,153.712
C04956=1076.193,-53.310,-57.688,173.265,21.073,153.712
C04957=1076.188,-53.559,-57.676,173.262,21.071,153.712
C04958=1076.182,-53.809,-57.664,173.261,21.069,153.712
C04959=1076.175,-54.059,-57.653,173.260,21.067,153.712
C04960=1076.170,-54.308,-57.641,173.258,21.065,153.712
C04961=1076.163,-54.558,-57.629,173.257,21.064,153.712
C04962=1076.157,-54.808,-57.617,173.255,21.062,153.711
C04963=1076.152,-55.057,-57.605,173.254,21.060,153.711
C04964=1076.145,-55.307,-57.593,173.253,21.058,153.711
C04965=1076.139,-55.557,-57.582,173.251,21.056,153.711
C04966=1076.133,-55.806,-57.570,173.250,21.054,153.711
C04967=1076.127,-56.056,-57.558,173.249,21.052,153.711
C04968=1076.120,-56.306,-57.547,173.247,21.051,153.711
C04969=1076.114,-56.555,-57.535,173.245,21.048,153.711
C04970=1076.109,-56.805,-57.523,173.244,21.046,153.710
C04971=1076.103,-57.054,-57.512,173.242,21.045,153.710
C04972=1076.096,-57.304,-57.500,173.241,21.043,153.710
C04973=1076.090,-57.554,-57.488,173.239,21.041,153.710
C04974=1076.084,-57.803,-57.476,173.238,21.039,153.710
C04975=1076.078,-58.053,-57.465,173.236,21.038,153.710
C04976=1076.072,-58.302,-57.453,173.235,21.036,153.710
C04977=1076.066,-58.553,-57.441,173.234,21.034,153.710
C04978=1076.060,-58.802,-57.430,173.232,21.032,153.710
C04979=1076.054,-59.052,-57.419,173.231,21.030,153.709
C04980=1076.047,-59.301,-57.407,173.230,21.028,153.709
C04981=1076.042,-59.551,-57.395,173.228,21.027,153.709
C04982=1076.036,-59.801,-57.383,173.226,21.025,153.709
C04983=1076.030,-60.050,-57.372,173.225,21.023,153.709
C04984=1076.023,-60.300,-57.360,173.223,21.021,153.709
C04985=1076.018,-60.550,-57.349,173.222,21.019,153.709
C04986=1076.012,-60.799,-57.337,173.220,21.017,153.709
C04987=1076.005,-61.049,-57.326,173.219,21.016,153.709
C04988=1075.999,-61.298,-57.314,173.217,21.014,153.708
C04989=1075.994,-61.549,-57.302,173.216,21.012,153.708
C04990=1075.988,-61.798,-57.291,173.215,21.010,153.708
C04991=1075.981,-62.048,-57.279,173.213,21.008,153.708
C04992=1075.975,-62.297,-57.268,173.212,21.007,153.708
C04993=1075.970,-62.547,-57.256,173.210,21.005,153.708
C04994=1075.964,-62.797,-57.245,173.209,21.003,153.708
C04995=1075.957,-63.046,-57.233,173.208,21.002,153.708
C04996=1075.951,-63.296,-57.222,173.205,20.999,153.708
C04997=1075.946,-63.546,-57.210,173.204,20.997,153.707
C04998=1075.940,-63.795,-57.199,173.202,20.996,153.707
C04999=1075.933,-64.045,-57.188,173.201,20.994,153.707
C05000=1075.927,-64.294,-57.176,173.200,20.992,153.707
C05001=1075.921,-64.544,-57.165,173.198,20.991,153.707
C05002=1075.916,-64.794,-57.153,173.197,20.989,153.707
C05003=1075.909,-65.044,-57.141,173.195,20.987,153.707
C05004=1075.903,-65.320,-57.129,173.194,20.985,153.707
C05005=1075.897,-65.596,-57.116,173.192,20.983,153.707
C05006=1075.889,-65.873,-57.104,173.191,20.981,153.706
C05007=1075.883,-66.149,-57.092,173.189,20.979,153.706
C05008=1075.878,-66.399,-57.080,173.188,20.977,153.706
C05009=1075.871,-66.649,-57.068,173.186,20.975,153.706
C05010=1075.866,-66.898,-57.057,173.185,20.974,153.706
C05011=1075.859,-67.148,-57.045,173.183,20.972,153.706
C05012=1075.853,-67.397,-57.035,173.182,20.971,153.706
C05013=1075.847,-67.647,-57.023,173.181,20.969,153.706
C05014=1075.842,-67.897,-57.012,173.178,20.967,153.706
C05015=1075.835,-68.147,-57.000,173.177,20.965,153.706
C05016=1075.829,-68.396,-56.989,173.176,20.963,153.706
C05017=1075.824,-68.646,-56.978,173.174,20.961,153.705
C05018=1075.817,-68.896,-56.967,173.173,20.959,153.705
C05019=1075.811,-69.145,-56.955,173.171,20.958,153.705
C05020=1075.806,-69.395,-56.943,173.170,20.956,153.705
C05021=1075.800,-69.645,-56.933,173.168,20.955,153.705
C05022=1075.794,-69.894,-56.922,173.167,20.953,153.705
C05023=1075.788,-70.144,-56.910,173.165,20.951,153.705
C05024=1075.782,-70.393,-56.899,173.164,20.949,153.705
C05025=1075.776,-70.643,-56.888,173.163,20.948,153.705
C05026=1075.770,-70.893,-56.877,173.161,20.946,153.705
C05027=1075.764,-71.143,-56.866,173.160,20.944,153.705
C05028=1075.758,-71.392,-56.853,173.158,20.942,153.704
C05029=1075.752,-71.642,-56.842,173.157,20.941,153.704
C05030=1075.747,-71.891,-56.832,173.155,20.939,153.704
C05031=1075.740,-72.142,-56.820,173.154,20.938,153.704
C05032=1075.735,-72.391,-56.809,173.153,20.936,153.704
C05033=1075.729,-72.641,-56.799,173.151,20.934,153.704
C05034=1075.722,-72.891,-56.787,173.150,20.932,153.704
C05035=1075.716,-73.140,-56.776,173.148,20.931,153.704
C05036=1075.711,-73.389,-56.764,173.146,20.928,153.704
C05037=1075.705,-73.640,-56.753,173.145,20.927,153.704
C05038=1075.699,-73.889,-56.742,173.143,20.925,153.704
C05039=1075.694,-74.139,-56.731,173.142,20.923,153.704
C05040=1075.687,-74.389,-56.720,173.140,20.921,153.703
C05041=1075.681,-74.638,-56.709,173.139,20.920,153.703
C05042=1075.676,-74.888,-56.698,173.137,20.919,153.703
C05043=1075.669,-75.138,-56.688,173.136,20.917,153.703
C05044=1075.663,-75.387,-56.677,173.134,20.915,153.703
C05045=1075.657,-75.637,-56.665,173.133,20.914,153.703
C05046=1075.651,-75.886,-56.654,173.132,20.912,153.703
C05047=1075.645,-76.136,-56.643,173.130,20.910,153.703
C05048=1075.638,-76.386,-56.632,173.128,20.909,153.703
C05049=1075.633,-76.635,-56.621,173.127,20.907,153.703
C05050=1075.627,-76.885,-56.610,173.126,20.906,153.703
C05051=1075.621,-77.135,-56.599,173.124,20.904,153.703
C05052=1075.615,-77.385,-56.588,173.123,20.902,153.703
C05053=1075.608,-77.634,-56.578,173.121,20.901,153.703
C05054=1075.602,-77.884,-56.566,173.120,20.899,153.703
C05055=1075.596,-78.133,-56.555,173.118,20.898,153.703
C05056=1075.591,-78.383,-56.545,173.117,20.896,153.702
C05057=1075.584,-78.633,-56.533,173.115,20.894,153.702
C05058=1075.579,-78.883,-56.522,173.114,20.893,153.702
C05059=1075.573,-79.132,-56.512,173.112,20.891,153.702
C05060=1075.566,-79.382,-56.500,173.111,20.890,153.702
C05061=1075.560,-79.632,-56.491,173.109,20.888,153.702
C05062=1075.555,-79.882,-56.480,173.108,20.887,153.702
C05063=1075.548,-80.132,-56.469,173.106,20.885,153.702
C05064=1075.542,-80.381,-56.458,173.105,20.883,153.702
C05065=1075.536,-80.630,-56.448,173.103,20.882,153.702
C05066=1075.530,-80.881,-56.436,173.102,20.880,153.702
C05067=1075.524,-81.130,-56.425,173.100,20.879,153.702
C05068=1075.518,-81.382,-56.415,173.099,20.878,153.702
C05069=1075.512,-81.634,-56.404,173.097,20.876,153.702
C05070=1075.505,-81.887,-56.393,173.096,20.874,153.702
C05071=1075.499,-82.139,-56.382,173.094,20.873,153.702
C05072=1075.492,-82.388,-56.371,173.093,20.871,153.702
C05073=1075.487,-82.638,-56.361,173.091,20.870,153.702
C05074=1075.481,-82.888,-56.350,173.090,20.868,153.702
C05075=1075.474,-83.138,-56.340,173.088,20.867,153.702
C05076=1075.468,-83.387,-56.329,173.087,20.866,153.702
C05077=1075.462,-83.637,-56.318,173.085,20.864,153.702
C05078=1075.456,-83.886,-56.307,173.084,20.862,153.701
C05079=1075.450,-84.137,-56.297,173.082,20.861,153.701
C05080=1075.444,-84.386,-56.286,173.081,20.859,153.701
C05081=1075.437,-84.636,-56.276,173.079,20.858,153.701
C05082=1075.432,-84.885,-56.265,173.078,20.856,153.701
C05083=1075.426,-85.135,-56.254,173.076,20.855,153.701
C05084=1075.419,-85.385,-56.243,173.075,20.854,153.701
C05085=1075.413,-85.635,-56.233,173.073,20.852,153.701
C05086=1075.407,-85.884,-56.223,173.072,20.851,153.701
C05087=1075.401,-86.134,-56.212,173.070,20.849,153.701
C05088=1075.395,-86.384,-56.201,173.069,20.848,153.701
C05089=1075.389,-86.634,-56.191,173.067,20.846,153.701
C05090=1075.383,-86.883,-56.180,173.065,20.845,153.701
C05091=1075.377,-87.132,-56.169,173.064,20.844,153.701
C05092=1075.370,-87.382,-56.159,173.063,20.842,153.701
C05093=1075.365,-87.632,-56.149,173.061,20.840,153.701
C05094=1075.358,-87.882,-56.138,173.060,20.839,153.701
C05095=1075.352,-88.131,-56.127,173.058,20.837,153.701
C05096=1075.347,-88.381,-56.117,173.056,20.836,153.701
C05097=1075.340,-88.631,-56.107,173.055,20.834,153.701
C05098=1075.334,-88.881,-56.096,173.053,20.833,153.701
C05099=1075.328,-89.130,-56.085,173.052,20.832,153.701
C05100=1075.322,-89.380,-56.075,173.050,20.830,153.701
C05101=1075.316,-89.630,-56.064,173.049,20.829,153.701
C05102=1075.309,-89.879,-56.054,173.047,20.827,153.701
C05103=1075.304,-90.129,-56.044,173.046,20.826,153.701
C05104=1075.297,-90.406,-56.032,173.044,20.824,153.701
C05105=1075.291,-90.681,-56.021,173.042,20.823,153.701
C05106=1075.284,-90.958,-56.009,173.040,20.821,153.701
C05107=1075.277,-91.233,-55.997,173.039,20.820,153.701
C05108=1075.271,-91.483,-55.987,173.037,20.818,153.701
C05109=1075.265,-91.732,-55.977,173.036,20.817,153.701
C05110=1075.259,-91.983,-55.966,173.034,20.815,153.701
C05111=1075.253,-92.232,-55.956,173.033,20.814,153.701
C05112=1075.247,-92.482,-55.945,173.031,20.812,153.701
C05113=1075.241,-92.732,-55.935,173.030,20.811,153.701
C05114=1075.235,-92.981,-55.925,173.028,20.810,153.701
C05115=1075.229,-93.231,-55.914,173.026,20.808,153.701
C05116=1075.223,-93.481,-55.904,173.025,20.807,153.700
C05117=1075.217,-93.731,-55.894,173.023,20.806,153.701
C05118=1075.211,-93.980,-55.884,173.022,20.804,153.701
C05119=1075.205,-94.230,-55.872,173.020,20.803,153.701
C05120=1075.198,-94.480,-55.863,173.019,20.802,153.701
C05121=1075.193,-94.729,-55.852,173.017,20.800,153.701
C05122=1075.187,-94.979,-55.842,173.016,20.799,153.701
C05123=1075.181,-95.229,-55.831,173.014,20.797,153.700
C05124=1075.175,-95.479,-55.821,173.012,20.796,153.700
C05125=1075.169,-95.728,-55.811,173.011,20.794,153.700
C05126=1075.163,-95.978,-55.801,173.010,20.793,153.700
C05127=1075.157,-96.227,-55.791,173.009,20.793,153.700
C05128=1075.151,-96.477,-55.780,173.007,20.791,153.700
C05129=1075.144,-96.727,-55.770,173.005,20.790,153.700
C05130=1075.139,-96.977,-55.760,173.004,20.788,153.700
C05131=1075.132,-97.226,-55.749,173.002,20.787,153.700
C05132=1075.126,-97.507,-55.738,173.001,20.785,153.700
C05133=1075.119,-97.788,-55.727,172.998,20.783,153.700
C05134=1075.112,-98.069,-55.716,172.997,20.782,153.700
C05135=1075.106,-98.350,-55.704,172.995,20.781,153.701
C05136=1075.099,-98.600,-55.694,172.994,20.780,153.700
C05137=1075.093,-98.850,-55.683,172.992,20.778,153.700
C05138=1075.087,-99.099,-55.673,172.991,20.777,153.700
C05139=1075.081,-99.349,-55.663,172.989,20.776,153.701
C05140=1075.074,-99.598,-55.654,172.987,20.775,153.701
C05141=1075.069,-99.848,-55.643,172.986,20.773,153.701
C05142=1075.063,-100.098,-55.633,172.984,20.772,153.701
C05143=1075.056,-100.347,-55.624,172.982,20.771,153.701
C05144=1075.051,-100.598,-55.613,172.981,20.769,153.701
C05145=1075.045,-100.847,-55.603,172.979,20.768,153.701
C05146=1075.038,-101.097,-55.593,172.978,20.767,153.701
C05147=1075.032,-101.347,-55.582,172.977,20.766,153.701
C05148=1075.026,-101.596,-55.573,172.975,20.765,153.701
C05149=1075.020,-101.846,-55.563,172.974,20.764,153.701
C05150=1075.014,-102.096,-55.552,172.972,20.762,153.701
C05151=1075.008,-102.346,-55.543,172.971,20.761,153.701
C05152=1075.002,-102.595,-55.533,172.969,20.760,153.701
C05153=1074.995,-102.845,-55.523,172.967,20.758,153.701
C05154=1074.990,-103.095,-55.513,172.966,20.757,153.701
C05155=1074.983,-103.344,-55.503,172.964,20.756,153.701
C05156=1074.977,-103.594,-55.493,172.963,20.755,153.701
C05157=1074.971,-103.843,-55.483,172.961,20.754,153.701
C05158=1074.965,-104.094,-55.473,172.959,20.752,153.701
C05159=1074.959,-104.343,-55.464,172.958,20.751,153.701
C05160=1074.953,-104.593,-55.453,172.956,20.750,153.701
C05161=1074.947,-104.843,-55.443,172.954,20.749,153.701
C05162=1074.941,-105.092,-55.434,172.954,20.748,153.701
C05163=1074.935,-105.342,-55.424,172.952,20.747,153.701
C05164=1074.928,-105.591,-55.414,172.951,20.745,153.701
C05165=1074.922,-105.841,-55.404,172.949,20.744,153.701
C05166=1074.917,-106.091,-55.394,172.947,20.743,153.701
C05167=1074.911,-106.341,-55.384,172.946,20.742,153.701
C05168=1074.904,-106.590,-55.374,172.944,20.741,153.701
C05169=1074.898,-106.840,-55.365,172.942,20.740,153.701
C05170=1074.893,-107.090,-55.354,172.941,20.738,153.701
C05171=1074.886,-107.340,-55.345,172.939,20.737,153.701
C05172=1074.880,-107.590,-55.335,172.937,20.736,153.701
C05173=1074.874,-107.839,-55.325,172.936,20.735,153.702
C05174=1074.868,-108.089,-55.315,172.934,20.734,153.702
C05175=1074.861,-108.339,-55.306,172.933,20.733,153.702
C05176=1074.855,-108.588,-55.296,172.932,20.732,153.702
C05177=1074.849,-108.838,-55.287,172.930,20.731,153.702
C05178=1074.844,-109.088,-55.277,172.928,20.729,153.702
C05179=1074.837,-109.337,-55.266,172.927,20.729,153.702
C05180=1074.831,-109.587,-55.257,172.925,20.727,153.702
C05181=1074.825,-109.837,-55.247,172.923,20.726,153.702
C05182=1074.819,-110.087,-55.238,172.922,20.725,153.702
C05183=1074.813,-110.337,-55.228,172.920,20.724,153.702
C05184=1074.806,-110.586,-55.219,172.918,20.723,153.702
C05185=1074.800,-110.836,-55.209,172.917,20.722,153.702
C05186=1074.794,-111.086,-55.199,172.916,20.721,153.702
C05187=1074.788,-111.336,-55.190,172.914,20.720,153.702
C05188=1074.781,-111.585,-55.180,172.913,20.719,153.702
C05189=1074.776,-111.835,-55.169,172.911,20.718,153.702
C05190=1074.770,-112.085,-55.160,172.909,20.717,153.702
C05191=1074.764,-112.335,-55.150,172.908,20.716,153.702
C05192=1074.757,-112.585,-55.141,172.906,20.714,153.702
C05193=1074.751,-112.834,-55.131,172.904,20.713,153.703
C05194=1074.745,-113.084,-55.122,172.903,20.712,153.703
C05195=1074.739,-113.334,-55.112,172.901,20.711,153.703
C05196=1074.732,-113.612,-55.101,172.899,20.710,153.703
C05197=1074.725,-113.890,-55.091,172.898,20.709,153.703
C05198=1074.718,-114.169,-55.081,172.896,20.708,153.703
C05199=1074.712,-114.447,-55.069,172.894,20.707,153.703
C05200=1074.706,-114.696,-55.059,172.893,20.705,153.703
C05201=1074.700,-114.946,-55.050,172.891,20.705,153.703
C05202=1074.694,-115.195,-55.040,172.889,20.704,153.703
C05203=1074.688,-115.445,-55.031,172.888,20.703,153.703
C05204=1074.681,-115.695,-55.022,172.887,20.702,153.703
C05205=1074.675,-115.944,-55.012,172.885,20.701,153.703
C05206=1074.669,-116.195,-55.004,172.883,20.700,153.704
C05207=1074.663,-116.445,-54.994,172.882,20.699,153.704
C05208=1074.656,-116.694,-54.984,172.880,20.698,153.704
C05209=1074.650,-116.944,-54.975,172.878,20.697,153.704
C05210=1074.644,-117.194,-54.965,172.877,20.696,153.704
C05211=1074.638,-117.444,-54.956,172.875,20.695,153.704
C05212=1074.632,-117.693,-54.946,172.873,20.694,153.704
C05213=1074.626,-117.943,-54.937,172.873,20.693,153.704
C05214=1074.620,-118.192,-54.927,172.871,20.692,153.704
C05215=1074.614,-118.442,-54.918,172.869,20.691,153.704
C05216=1074.608,-118.692,-54.908,172.868,20.690,153.704
C05217=1074.602,-118.942,-54.899,172.866,20.689,153.704
C05218=1074.595,-119.192,-54.889,172.864,20.688,153.704
C05219=1074.589,-119.442,-54.881,172.862,20.687,153.705
C05220=1074.583,-119.691,-54.872,172.861,20.686,153.705
C05221=1074.577,-119.941,-54.862,172.860,20.686,153.705
C05222=1074.571,-120.190,-54.852,172.858,20.685,153.705
C05223=1074.565,-120.440,-54.843,172.856,20.684,153.705
C05224=1074.559,-120.690,-54.833,172.855,20.683,153.705
C05225=1074.552,-120.940,-54.824,172.853,20.682,153.705
C05226=1074.546,-121.190,-54.815,172.851,20.681,153.705
C05227=1074.540,-121.439,-54.806,172.849,20.680,153.705
C05228=1074.534,-121.689,-54.797,172.849,20.680,153.705
C05229=1074.528,-121.939,-54.787,172.847,20.679,153.706
C05230=1074.522,-122.188,-54.778,172.845,20.677,153.706
C05231=1074.515,-122.438,-54.768,172.844,20.676,153.706
C05232=1074.510,-122.689,-54.759,172.842,20.676,153.706
C05233=1074.503,-122.937,-54.751,172.840,20.675,153.706
C05234=1074.497,-123.187,-54.741,172.838,20.674,153.706
C05235=1074.491,-123.437,-54.731,172.837,20.673,153.706
C05236=1074.485,-123.687,-54.723,172.836,20.672,153.706
C05237=1074.479,-123.937,-54.713,172.834,20.672,153.706
C05238=1074.473,-124.187,-54.703,172.832,20.671,153.706
C05239=1074.466,-124.436,-54.695,172.830,20.670,153.707
C05240=1074.461,-124.686,-54.686,172.829,20.669,153.707
C05241=1074.454,-124.936,-54.676,172.827,20.668,153.707
C05242=1074.448,-125.186,-54.667,172.826,20.668,153.707
C05243=1074.441,-125.435,-54.658,172.824,20.667,153.707
C05244=1074.436,-125.685,-54.649,172.823,20.666,153.707
C05245=1074.430,-125.935,-54.640,172.821,20.665,153.707
C05246=1074.424,-126.185,-54.630,172.819,20.664,153.707
C05247=1074.417,-126.434,-54.621,172.817,20.663,153.707
C05248=1074.411,-126.685,-54.612,172.816,20.662,153.708
C05249=1074.405,-126.934,-54.603,172.815,20.662,153.708
C05250=1074.398,-127.183,-54.594,172.813,20.661,153.708
C05251=1074.393,-127.434,-54.585,172.811,20.660,153.708
C05252=1074.386,-127.683,-54.576,172.809,20.659,153.708
C05253=1074.380,-127.935,-54.567,172.808,20.658,153.708
C05254=1074.376,-128.185,-54.557,172.806,20.657,153.708
C05255=1074.374,-128.436,-54.546,172.805,20.655,153.708
C05256=1074.374,-128.690,-54.535,172.804,20.652,153.707
C05257=1074.376,-128.943,-54.522,172.803,20.648,153.707
C05258=1074.382,-129.195,-54.509,172.803,20.643,153.706
C05259=1074.389,-129.446,-54.494,172.803,20.638,153.705
C05260=1073.995,-129.467,-54.650,172.758,20.770,153.737
C05261=1073.988,-129.217,-54.664,172.758,20.775,153.738
C05262=1073.983,-128.964,-54.678,172.758,20.780,153.738
C05263=1073.980,-128.711,-54.691,172.759,20.784,153.739
C05264=1073.979,-128.457,-54.703,172.759,20.787,153.739
C05265=1073.981,-128.207,-54.714,172.761,20.789,153.740
C05266=1073.986,-127.956,-54.724,172.762,20.790,153.740
C05267=1073.992,-127.706,-54.733,172.764,20.791,153.739
C05268=1073.998,-127.456,-54.742,172.766,20.792,153.739
C05269=1074.004,-127.206,-54.751,172.768,20.793,153.739
C05270=1074.010,-126.956,-54.759,172.769,20.794,153.739
C05271=1074.017,-126.706,-54.769,172.770,20.794,153.739
C05272=1074.023,-126.457,-54.778,172.772,20.795,153.739
C05273=1074.029,-126.207,-54.787,172.774,20.796,153.739
C05274=1074.035,-125.957,-54.796,172.775,20.797,153.739
C05275=1074.041,-125.707,-54.806,172.777,20.798,153.739
C05276=1074.048,-125.458,-54.815,172.779,20.798,153.738
C05277=1074.053,-125.208,-54.823,172.781,20.799,153.738
C05278=1074.059,-124.958,-54.833,172.782,20.800,153.738
C05279=1074.066,-124.708,-54.842,172.783,20.801,153.738
C05280=1074.072,-124.459,-54.851,172.785,20.801,153.738
C05281=1074.078,-124.208,-54.860,172.787,20.802,153.738
C05282=1074.085,-123.959,-54.870,172.789,20.803,153.738
C05283=1074.090,-123.709,-54.879,172.790,20.804,153.738
C05284=1074.096,-123.460,-54.888,172.792,20.805,153.738
C05285=1074.103,-123.210,-54.897,172.793,20.806,153.738
C05286=1074.109,-122.960,-54.906,172.794,20.807,153.737
C05287=1074.115,-122.710,-54.916,172.796,20.808,153.737
C05288=1074.121,-122.461,-54.925,172.798,20.809,153.737
C05289=1074.127,-122.211,-54.935,172.800,20.810,153.737
C05290=1074.133,-121.961,-54.944,172.801,20.810,153.737
C05291=1074.140,-121.711,-54.952,172.803,20.811,153.737
C05292=1074.146,-121.461,-54.962,172.805,20.812,153.737
C05293=1074.152,-121.212,-54.972,172.806,20.813,153.737
C05294=1074.158,-120.962,-54.981,172.807,20.814,153.737
C05295=1074.164,-120.713,-54.990,172.809,20.815,153.737
C05296=1074.170,-120.463,-55.000,172.811,20.816,153.736
C05297=1074.176,-120.212,-55.009,172.813,20.817,153.736
C05298=1074.182,-119.963,-55.018,172.814,20.818,153.736
C05299=1074.189,-119.713,-55.027,172.816,20.818,153.736
C05300=1074.195,-119.463,-55.037,172.817,20.819,153.736
C05301=1074.201,-119.214,-55.046,172.819,20.820,153.736
C05302=1074.207,-118.964,-55.056,172.820,20.821,153.736
C05303=1074.213,-118.715,-55.065,172.822,20.822,153.736
C05304=1074.219,-118.465,-55.075,172.824,20.823,153.736
C05305=1074.225,-118.214,-55.084,172.825,20.824,153.736
C05306=1074.231,-117.965,-55.093,172.827,20.825,153.736
C05307=1074.237,-117.715,-55.103,172.829,20.826,153.736
C05308=1074.244,-117.465,-55.112,172.831,20.827,153.735
C05309=1074.250,-117.215,-55.122,172.831,20.828,153.735
C05310=1074.257,-116.966,-55.131,172.833,20.829,153.735
C05311=1074.262,-116.717,-55.140,172.835,20.830,153.735
C05312=1074.268,-116.467,-55.150,172.836,20.831,153.735
C05313=1074.275,-116.217,-55.159,172.838,20.832,153.735
C05314=1074.281,-115.967,-55.169,172.840,20.833,153.735
C05315=1074.287,-115.717,-55.178,172.841,20.834,153.735
C05316=1074.293,-115.468,-55.188,172.843,20.835,153.735
C05317=1074.299,-115.218,-55.197,172.845,20.836,153.735
C05318=1074.305,-114.968,-55.207,172.846,20.837,153.735
C05319=1074.312,-114.718,-55.217,172.847,20.837,153.735
C05320=1074.318,-114.468,-55.226,172.849,20.839,153.735
C05321=1074.325,-114.190,-55.237,172.851,20.840,153.735
C05322=1074.331,-113.912,-55.248,172.852,20.841,153.734
C05323=1074.338,-113.633,-55.258,172.855,20.843,153.734
C05324=1074.344,-113.355,-55.269,172.857,20.843,153.734
C05325=1074.351,-113.105,-55.278,172.858,20.845,153.734
C05326=1074.357,-112.856,-55.288,172.860,20.846,153.734
C05327=1074.363,-112.606,-55.297,172.861,20.846,153.734
C05328=1074.369,-112.356,-55.307,172.862,20.848,153.734
C05329=1074.375,-112.106,-55.316,172.864,20.848,153.734
C05330=1074.382,-111.856,-55.326,172.866,20.850,153.734
C05331=1074.388,-111.607,-55.336,172.867,20.851,153.734
C05332=1074.393,-111.357,-55.346,172.869,20.852,153.734
C05333=1074.400,-111.107,-55.356,172.871,20.853,153.734
C05334=1074.406,-110.857,-55.366,172.872,20.854,153.734
C05335=1074.412,-110.608,-55.375,172.874,20.855,153.734
C05336=1074.418,-110.358,-55.385,172.876,20.856,153.734
C05337=1074.424,-110.108,-55.394,172.876,20.857,153.734
C05338=1074.430,-109.859,-55.403,172.878,20.858,153.734
C05339=1074.436,-109.609,-55.413,172.880,20.860,153.734
C05340=1074.443,-109.360,-55.423,172.881,20.860,153.733
C05341=1074.449,-109.110,-55.433,172.883,20.861,153.733
C05342=1074.455,-108.860,-55.442,172.885,20.863,153.733
C05343=1074.460,-108.610,-55.453,172.886,20.864,153.733
C05344=1074.466,-108.361,-55.462,172.888,20.865,153.733
C05345=1074.473,-108.111,-55.472,172.890,20.866,153.733
C05346=1074.479,-107.862,-55.482,172.891,20.867,153.733
C05347=1074.486,-107.611,-55.492,172.893,20.868,153.733
C05348=1074.491,-107.362,-55.501,172.895,20.870,153.733
C05349=1074.498,-107.112,-55.511,172.896,20.871,153.733
C05350=1074.503,-106.862,-55.521,172.897,20.872,153.733
C05351=1074.510,-106.613,-55.531,172.898,20.873,153.733
C05352=1074.516,-106.363,-55.541,172.900,20.874,153.733
C05353=1074.522,-106.113,-55.550,172.902,20.875,153.733
C05354=1074.528,-105.863,-55.560,172.903,20.876,153.733
C05355=1074.534,-105.613,-55.570,172.905,20.878,153.733
C05356=1074.541,-105.363,-55.581,172.907,20.879,153.733
C05357=1074.547,-105.114,-55.590,172.908,20.880,153.733
C05358=1074.553,-104.864,-55.600,172.910,20.881,153.733
C05359=1074.559,-104.614,-55.611,172.912,20.882,153.733
C05360=1074.565,-104.365,-55.620,172.913,20.884,153.733
C05361=1074.571,-104.115,-55.630,172.915,20.885,153.733
C05362=1074.577,-103.865,-55.639,172.916,20.886,153.733
C05363=1074.583,-103.616,-55.650,172.918,20.887,153.733
C05364=1074.589,-103.366,-55.660,172.919,20.888,153.733
C05365=1074.595,-103.116,-55.669,172.920,20.889,153.732
C05366=1074.601,-102.866,-55.680,172.922,20.891,153.733
C05367=1074.607,-102.617,-55.690,172.923,20.892,153.733
C05368=1074.613,-102.367,-55.699,172.925,20.893,153.732
C05369=1074.620,-102.118,-55.710,172.927,20.894,153.732
C05370=1074.625,-101.868,-55.720,172.928,20.896,153.732
C05371=1074.631,-101.618,-55.729,172.930,20.897,153.732
C05372=1074.638,-101.369,-55.740,172.932,20.898,153.732
C05373=1074.643,-101.118,-55.750,172.933,20.900,153.732
C05374=1074.649,-100.869,-55.759,172.935,20.901,153.732
C05375=1074.656,-100.619,-55.770,172.936,20.902,153.732
C05376=1074.661,-100.369,-55.780,172.938,20.903,153.732
C05377=1074.668,-100.119,-55.790,172.940,20.904,153.732
C05378=1074.675,-99.870,-55.800,172.941,20.906,153.732
C05379=1074.681,-99.620,-55.810,172.943,20.907,153.732
C05380=1074.687,-99.370,-55.821,172.944,20.909,153.732
C05381=1074.693,-99.121,-55.830,172.946,20.909,153.732
C05382=1074.699,-98.871,-55.840,172.948,20.911,153.732
C05383=1074.705,-98.621,-55.851,172.948,20.912,153.732
C05384=1074.711,-98.372,-55.860,172.950,20.913,153.732
C05385=1074.718,-98.090,-55.872,172.952,20.915,153.732
C05386=1074.725,-97.809,-55.883,172.954,20.916,153.732
C05387=1074.732,-97.529,-55.894,172.955,20.917,153.732
C05388=1074.738,-97.248,-55.906,172.957,20.919,153.732
C05389=1074.745,-96.998,-55.917,172.959,20.920,153.732
C05390=1074.751,-96.748,-55.927,172.960,20.922,153.732
C05391=1074.757,-96.499,-55.937,172.962,20.923,153.732
C05392=1074.762,-96.248,-55.947,172.963,20.925,153.732
C05393=1074.769,-95.999,-55.957,172.965,20.926,153.732
C05394=1074.774,-95.749,-55.968,172.966,20.927,153.732
C05395=1074.780,-95.500,-55.979,172.968,20.928,153.732
C05396=1074.786,-95.250,-55.988,172.970,20.930,153.732
C05397=1074.792,-95.000,-55.999,172.971,20.931,153.732
C05398=1074.798,-94.751,-56.009,172.973,20.933,153.732
C05399=1074.804,-94.501,-56.019,172.974,20.934,153.732
C05400=1074.811,-94.251,-56.029,172.976,20.935,153.732
C05401=1074.816,-94.001,-56.040,172.977,20.937,153.732
C05402=1074.823,-93.752,-56.051,172.979,20.938,153.732
C05403=1074.828,-93.502,-56.061,172.980,20.940,153.732
C05404=1074.835,-93.253,-56.071,172.982,20.941,153.732
C05405=1074.840,-93.002,-56.081,172.983,20.943,153.732
C05406=1074.846,-92.753,-56.092,172.985,20.944,153.732
C05407=1074.853,-92.502,-56.102,172.986,20.945,153.732
C05408=1074.859,-92.253,-56.113,172.988,20.947,153.732
C05409=1074.865,-92.004,-56.123,172.990,20.948,153.732
C05410=1074.870,-91.754,-56.133,172.991,20.950,153.732
C05411=1074.877,-91.505,-56.144,172.993,20.951,153.732
C05412=1074.882,-91.254,-56.154,172.994,20.953,153.732
C05413=1074.889,-91.005,-56.164,172.996,20.954,153.732
C05414=1074.895,-90.755,-56.175,172.997,20.955,153.732
C05415=1074.901,-90.505,-56.185,172.999,20.957,153.733
C05416=1074.907,-90.256,-56.196,173.000,20.958,153.733
C05417=1074.913,-90.006,-56.207,173.001,20.959,153.733
C05418=1074.919,-89.756,-56.216,173.003,20.961,153.733
C05419=1074.925,-89.506,-56.227,173.004,20.962,153.733
C05420=1074.931,-89.257,-56.238,173.006,20.964,153.733
C05421=1074.937,-89.007,-56.248,173.007,20.965,153.733
C05422=1074.943,-88.758,-56.259,173.009,20.966,153.733
C05423=1074.949,-88.508,-56.269,173.010,20.968,153.733
C05424=1074.956,-88.258,-56.280,173.012,20.969,153.733
C05425=1074.961,-88.008,-56.290,173.013,20.971,153.733
C05426=1074.968,-87.759,-56.301,173.015,20.972,153.733
C05427=1074.973,-87.509,-56.312,173.016,20.974,153.733
C05428=1074.980,-87.259,-56.321,173.018,20.975,153.733
C05429=1074.986,-87.009,-56.332,173.019,20.976,153.733
C05430=1074.992,-86.760,-56.343,173.021,20.978,153.733
C05431=1074.998,-86.511,-56.353,173.023,20.979,153.733
C05432=1075.004,-86.260,-56.364,173.024,20.981,153.733
C05433=1075.010,-86.010,-56.375,173.026,20.982,153.733
C05434=1075.016,-85.761,-56.385,173.027,20.984,153.733
C05435=1075.022,-85.512,-56.396,173.028,20.986,153.733
C05436=1075.028,-85.262,-56.407,173.030,20.987,153.733
C05437=1075.035,-85.012,-56.417,173.032,20.988,153.733
C05438=1075.040,-84.762,-56.428,173.033,20.990,153.733
C05439=1075.047,-84.513,-56.438,173.035,20.991,153.733
C05440=1075.053,-84.263,-56.449,173.036,20.993,153.733
C05441=1075.059,-84.013,-56.460,173.038,20.994,153.733
C05442=1075.065,-83.764,-56.470,173.039,20.996,153.733
C05443=1075.071,-83.513,-56.481,173.041,20.997,153.733
C05444=1075.077,-83.264,-56.492,173.042,20.999,153.733
C05445=1075.084,-83.015,-56.502,173.044,21.000,153.733
C05446=1075.090,-82.765,-56.513,173.045,21.002,153.733
C05447=1075.096,-82.515,-56.524,173.047,21.003,153.733
C05448=1075.102,-82.266,-56.535,173.048,21.005,153.734
C05449=1075.109,-81.987,-56.546,173.051,21.006,153.733
C05450=1075.115,-81.708,-56.559,173.052,21.008,153.734
